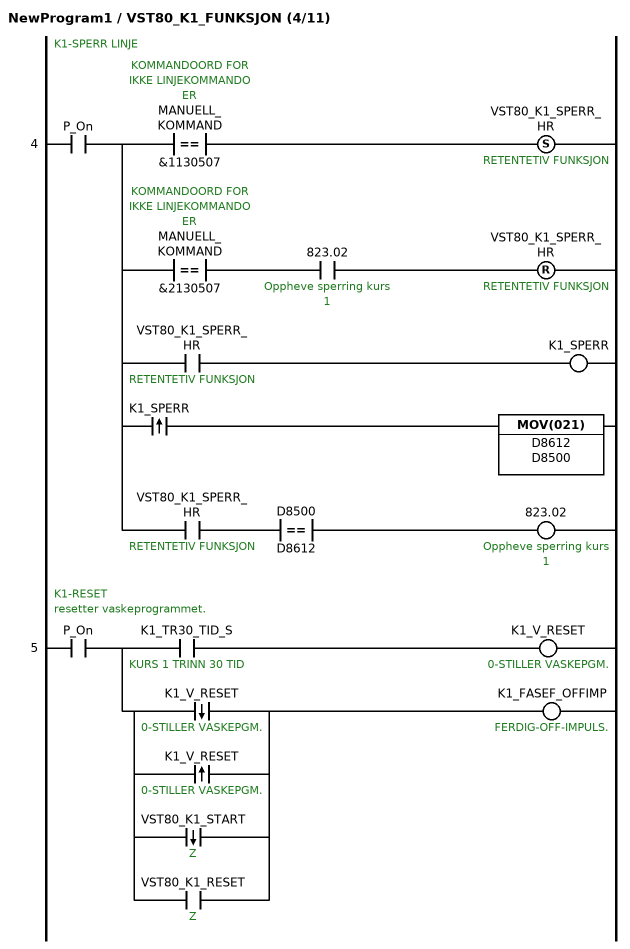
; [picture p120: NewProgram1 / VST80_K1_FUNKSJON, rungs 4-5]
; rung 4: K1-SPERR LINJE
LD P_On
OUT TR0
AND=L(301) MANUELL_KOMMAND &1130507  ; KOMMANDOORD FOR IKKE LINJEKOMMANDOER
SET VST80_K1_SPERR_HR  ; RETENTETIV FUNKSJON
LD TR0
AND=L(301) MANUELL_KOMMAND &2130507  ; KOMMANDOORD FOR IKKE LINJEKOMMANDOER
AND 823.02  ; Oppheve sperring kurs 1
RSET VST80_K1_SPERR_HR  ; RETENTETIV FUNKSJON
LD TR0
AND VST80_K1_SPERR_HR  ; RETENTETIV FUNKSJON
OUT K1_SPERR
LD TR0
@AND K1_SPERR
MOV(021) D8612 D8500
LD TR0
AND VST80_K1_SPERR_HR  ; RETENTETIV FUNKSJON
AND=(300) D8500 D8612
OUT 823.02  ; Oppheve sperring kurs 1
; rung 5: K1-RESET / resetter vaskeprogrammet.
LD P_On
OUT TR0
AND K1_TR30_TID_S  ; KURS 1 TRINN 30 TID
OUT K1_V_RESET  ; 0-STILLER VASKEPGM.
LD TR0
%LD K1_V_RESET  ; 0-STILLER VASKEPGM.
@OR K1_V_RESET  ; 0-STILLER VASKEPGM.
%OR VST80_K1_START  ; Z
OR VST80_K1_RESET  ; Z
ANDLD
OUT K1_FASEF_OFFIMP  ; FERDIG-OFF-IMPULS.

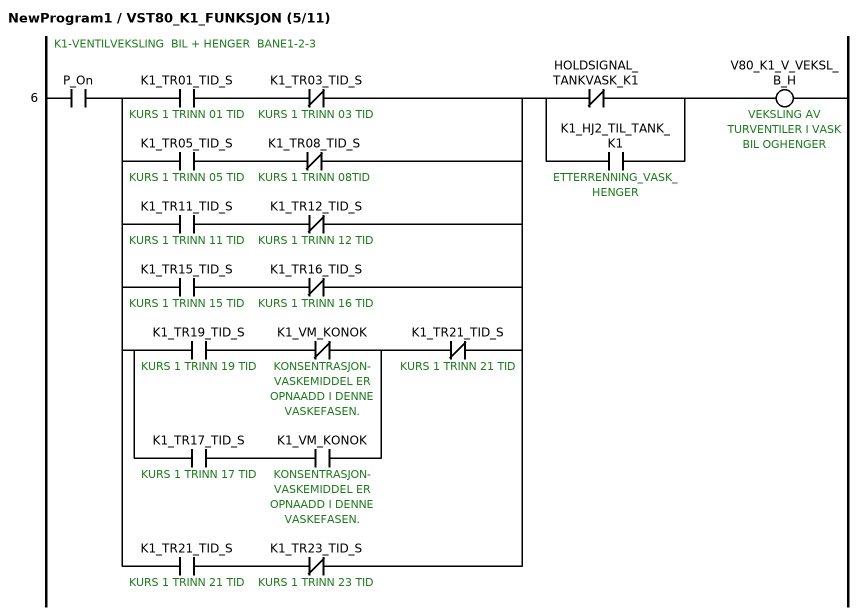
; rung 6: K1-VENTILVEKSLING  BIL + HENGER  BANE1-2-3
LD P_On
LD K1_TR01_TID_S  ; KURS 1 TRINN 01 TID
ANDNOT K1_TR03_TID_S  ; KURS 1 TRINN 03 TID
LD K1_TR05_TID_S  ; KURS 1 TRINN 05 TID
ANDNOT K1_TR08_TID_S  ; KURS 1 TRINN 08TID
ORLD
LD K1_TR11_TID_S  ; KURS 1 TRINN 11 TID
ANDNOT K1_TR12_TID_S  ; KURS 1 TRINN 12 TID
ORLD
LD K1_TR15_TID_S  ; KURS 1 TRINN 15 TID
ANDNOT K1_TR16_TID_S  ; KURS 1 TRINN 16 TID
ORLD
LD K1_TR19_TID_S  ; KURS 1 TRINN 19 TID
ANDNOT K1_VM_KONOK  ; KONSENTRASJON-VASKEMIDDEL ER OPNAADD I DENNE VASKEFASEN.
LD K1_TR17_TID_S  ; KURS 1 TRINN 17 TID
AND K1_VM_KONOK  ; KONSENTRASJON-VASKEMIDDEL ER OPNAADD I DENNE VASKEFASEN.
ORLD
ANDNOT K1_TR21_TID_S  ; KURS 1 TRINN 21 TID
ORLD
LD K1_TR21_TID_S  ; KURS 1 TRINN 21 TID
ANDNOT K1_TR23_TID_S  ; KURS 1 TRINN 23 TID
ORLD
ANDLD
LDNOT HOLDSIGNAL_TANKVASK_K1
OR K1_HJ2_TIL_TANK_K1  ; ETTERRENNING_VASK_HENGER
ANDLD
OUT V80_K1_V_VEKSL_B_H  ; VEKSLING AV TURVENTILER I VASK BIL OGHENGER

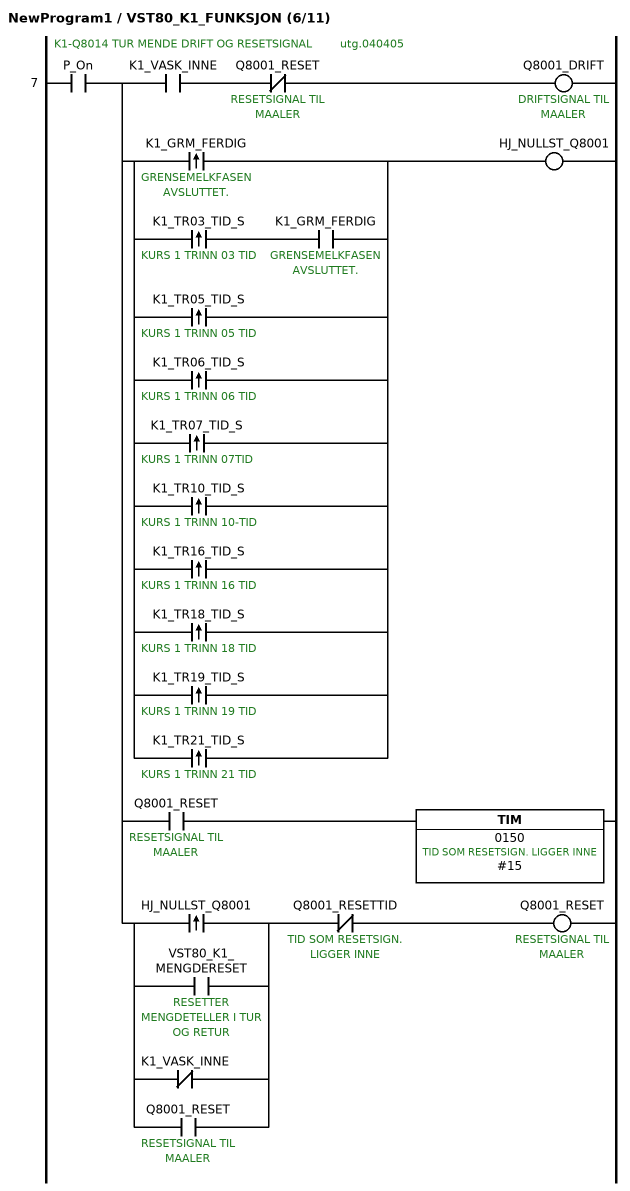
; rung 7: K1-Q8014 TUR MENDE DRIFT OG RESETSIGNAL        utg.040405
LD P_On
OUT TR0
AND K1_VASK_INNE
ANDNOT Q8001_RESET  ; RESETSIGNAL TIL MAALER
OUT Q8001_DRIFT  ; DRIFTSIGNAL TIL MAALER
LD TR0
@LD K1_GRM_FERDIG  ; GRENSEMELKFASEN AVSLUTTET.
@LD K1_TR03_TID_S  ; KURS 1 TRINN 03 TID
AND K1_GRM_FERDIG  ; GRENSEMELKFASEN AVSLUTTET.
ORLD
@OR K1_TR05_TID_S  ; KURS 1 TRINN 05 TID
@OR K1_TR06_TID_S  ; KURS 1 TRINN 06 TID
@OR K1_TR07_TID_S  ; KURS 1 TRINN 07TID
@OR K1_TR10_TID_S  ; KURS 1 TRINN 10-TID
@OR K1_TR16_TID_S  ; KURS 1 TRINN 16 TID
@OR K1_TR18_TID_S  ; KURS 1 TRINN 18 TID
@OR K1_TR19_TID_S  ; KURS 1 TRINN 19 TID
@OR K1_TR21_TID_S  ; KURS 1 TRINN 21 TID
ANDLD
OUT HJ_NULLST_Q8001
LD TR0
AND Q8001_RESET  ; RESETSIGNAL TIL MAALER
TIM 0150 #15  ; TID SOM RESETSIGN. LIGGER INNE
LD TR0
@LD HJ_NULLST_Q8001
OR VST80_K1_MENGDERESET  ; RESETTER MENGDETELLER I TUR OG RETUR
ORNOT K1_VASK_INNE
OR Q8001_RESET  ; RESETSIGNAL TIL MAALER
ANDLD
ANDNOT Q8001_RESETTID  ; TID SOM RESETSIGN. LIGGER INNE
OUT Q8001_RESET  ; RESETSIGNAL TIL MAALER

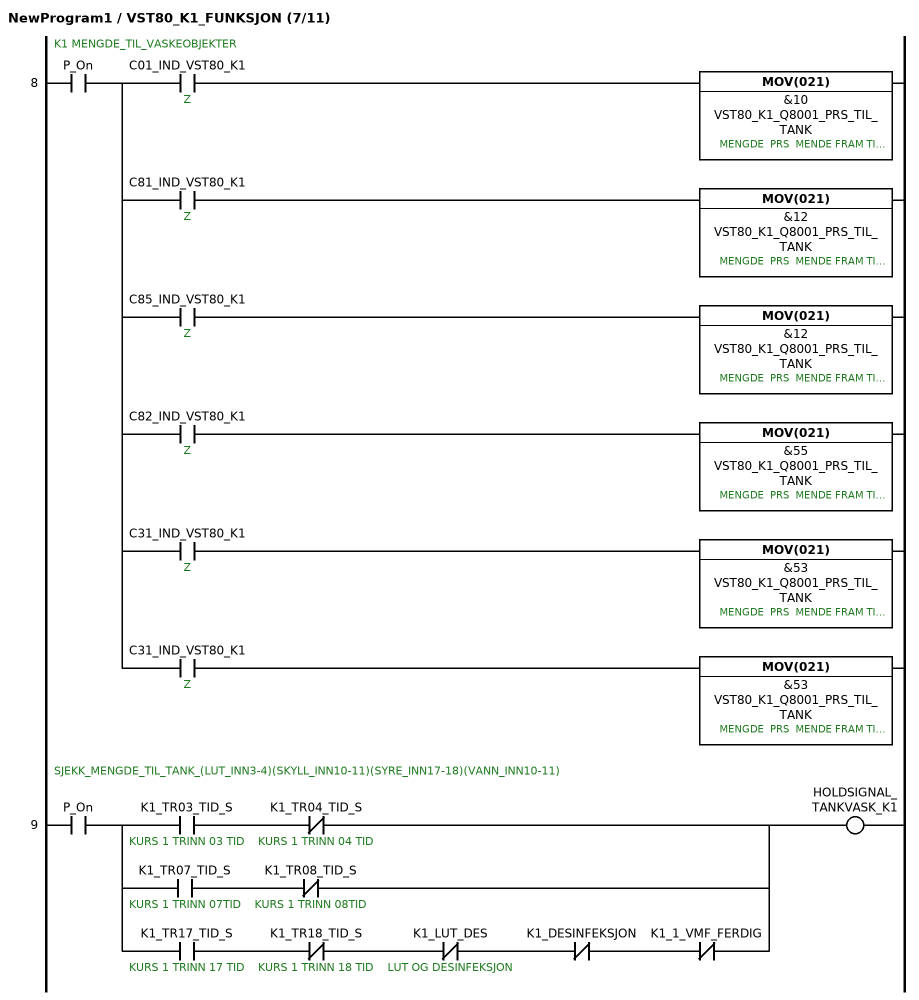
; rung 8: K1 MENGDE_TIL_VASKEOBJEKTER
LD P_On
OUT TR0
AND C01_IND_VST80_K1  ; Z
MOV(021) &10 VST80_K1_Q8001_PRS_TIL_TANK  ; MENGDE  PRS  MENDE FRAM TIL TANK
LD TR0
AND C81_IND_VST80_K1  ; Z
MOV(021) &12 VST80_K1_Q8001_PRS_TIL_TANK  ; MENGDE  PRS  MENDE FRAM TIL TANK
LD TR0
AND C85_IND_VST80_K1  ; Z
MOV(021) &12 VST80_K1_Q8001_PRS_TIL_TANK  ; MENGDE  PRS  MENDE FRAM TIL TANK
LD TR0
AND C82_IND_VST80_K1  ; Z
MOV(021) &55 VST80_K1_Q8001_PRS_TIL_TANK  ; MENGDE  PRS  MENDE FRAM TIL TANK
LD TR0
AND C31_IND_VST80_K1  ; Z
MOV(021) &53 VST80_K1_Q8001_PRS_TIL_TANK  ; MENGDE  PRS  MENDE FRAM TIL TANK
LD TR0
AND C31_IND_VST80_K1  ; Z
MOV(021) &53 VST80_K1_Q8001_PRS_TIL_TANK  ; MENGDE  PRS  MENDE FRAM TIL TANK
; rung 9: SJEKK_MENGDE_TIL_TANK_(LUT_INN3-4)(SKYLL_INN10-11)(SYRE_INN17-18)(VANN_INN10-11)
LD P_On
LD K1_TR03_TID_S  ; KURS 1 TRINN 03 TID
ANDNOT K1_TR04_TID_S  ; KURS 1 TRINN 04 TID
LD K1_TR07_TID_S  ; KURS 1 TRINN 07TID
ANDNOT K1_TR08_TID_S  ; KURS 1 TRINN 08TID
ORLD
LD K1_TR17_TID_S  ; KURS 1 TRINN 17 TID
ANDNOT K1_TR18_TID_S  ; KURS 1 TRINN 18 TID
ANDNOT K1_LUT_DES  ; LUT OG DESINFEKSJON
ANDNOT K1_DESINFEKSJON
ANDNOT K1_1_VMF_FERDIG
ORLD
ANDLD
OUT HOLDSIGNAL_TANKVASK_K1

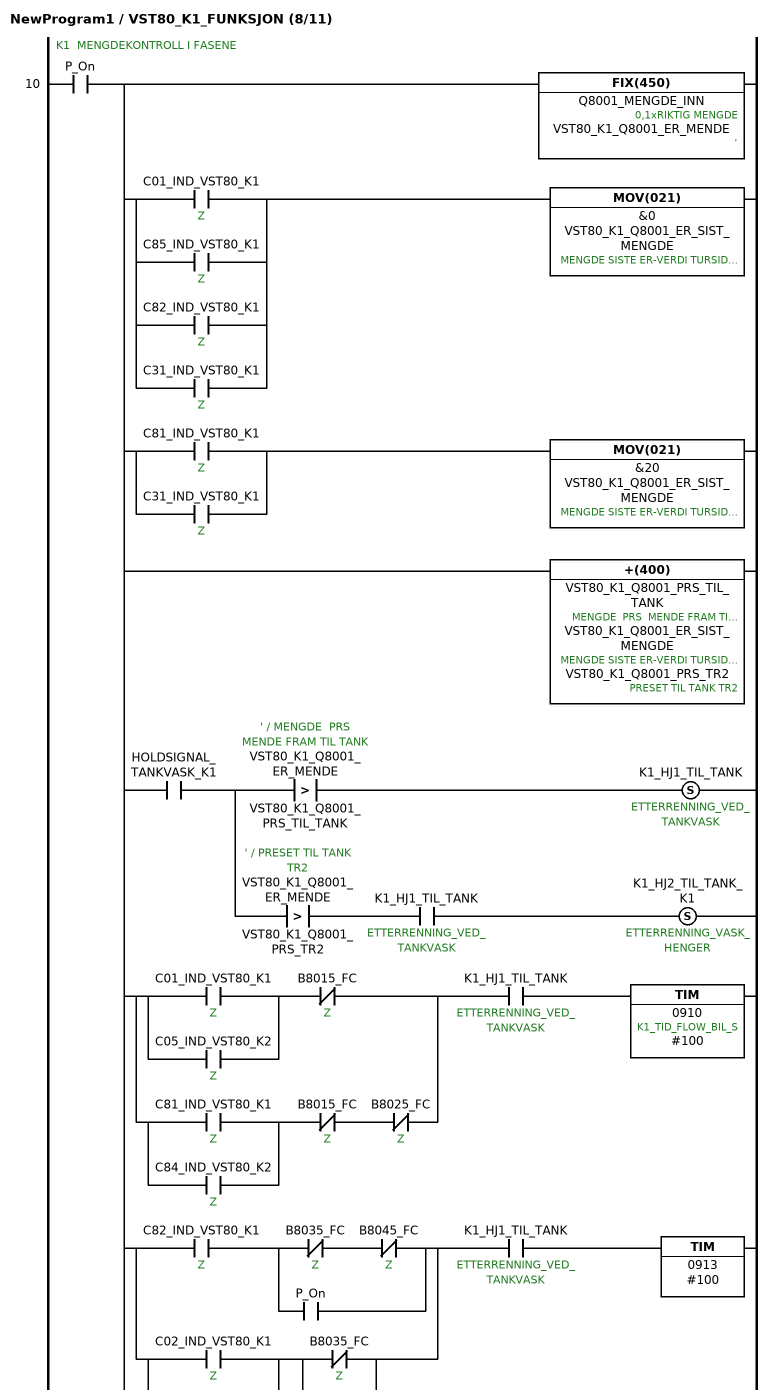

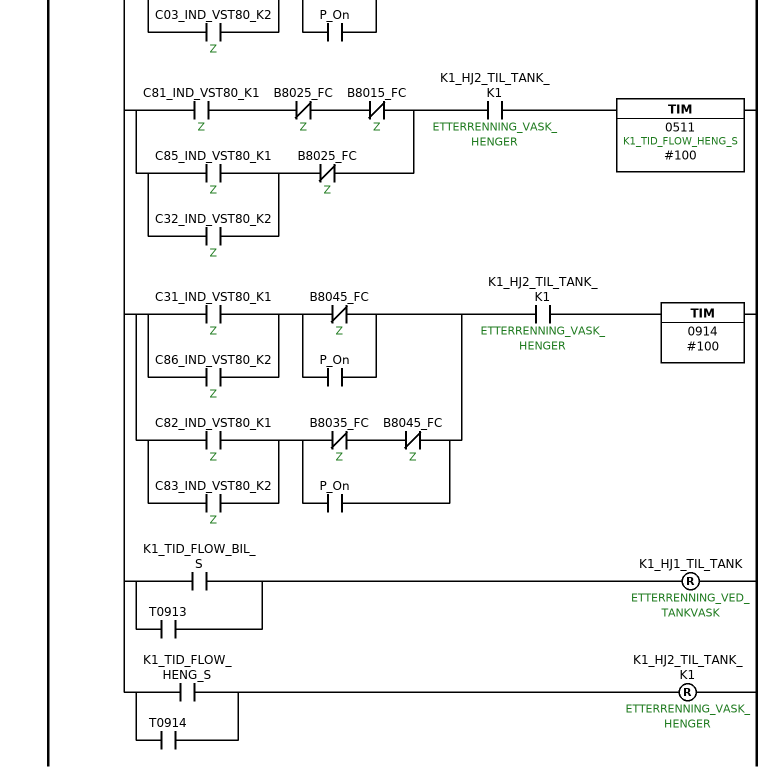
; rung 10: K1  MENGDEKONTROLL I FASENE
LD P_On
OUT TR0
FIX(450) Q8001_MENGDE_INN VST80_K1_Q8001_ER_MENDE  ; 0,1xRIKTIG MENGDE, '
LD C01_IND_VST80_K1  ; Z
OR C85_IND_VST80_K1  ; Z
OR C82_IND_VST80_K1  ; Z
OR C31_IND_VST80_K1  ; Z
ANDLD
MOV(021) &0 VST80_K1_Q8001_ER_SIST_MENGDE  ; MENGDE SISTE ER-VERDI TURSIDE PAA KURSEN
LD TR0
LD C81_IND_VST80_K1  ; Z
OR C31_IND_VST80_K1  ; Z
ANDLD
MOV(021) &20 VST80_K1_Q8001_ER_SIST_MENGDE  ; MENGDE SISTE ER-VERDI TURSIDE PAA KURSEN
LD TR0
+(400) VST80_K1_Q8001_PRS_TIL_TANK VST80_K1_Q8001_ER_SIST_MENGDE VST80_K1_Q8001_PRS_TR2  ; MENGDE  PRS  MENDE FRAM TIL TANK, MENGDE SISTE ER-VERDI TURSIDE PAA KURSEN, PRESET TIL TANK TR2
AND HOLDSIGNAL_TANKVASK_K1
OUT TR1
AND>(320) VST80_K1_Q8001_ER_MENDE VST80_K1_Q8001_PRS_TIL_TANK  ; ', MENGDE  PRS  MENDE FRAM TIL TANK
SET K1_HJ1_TIL_TANK  ; ETTERRENNING_VED_TANKVASK
LD TR1
AND>(320) VST80_K1_Q8001_ER_MENDE VST80_K1_Q8001_PRS_TR2  ; ', PRESET TIL TANK TR2
AND K1_HJ1_TIL_TANK  ; ETTERRENNING_VED_TANKVASK
SET K1_HJ2_TIL_TANK_K1  ; ETTERRENNING_VASK_HENGER
LD TR0
LD C01_IND_VST80_K1  ; Z
OR C05_IND_VST80_K2  ; Z
ANDNOT B8015_FC  ; Z
LD C81_IND_VST80_K1  ; Z
OR C84_IND_VST80_K2  ; Z
ANDNOT B8015_FC  ; Z
ANDNOT B8025_FC  ; Z
ORLD
ANDLD
AND K1_HJ1_TIL_TANK  ; ETTERRENNING_VED_TANKVASK
TIM 0910 #100  ; K1_TID_FLOW_BIL_S
LD TR0
LD C82_IND_VST80_K1  ; Z
LDNOT B8035_FC  ; Z
ANDNOT B8045_FC  ; Z
OR P_On
ANDLD
LD C02_IND_VST80_K1  ; Z
OR C03_IND_VST80_K2  ; Z
LDNOT B8035_FC  ; Z
OR P_On
ANDLD
ORLD
ANDLD
AND K1_HJ1_TIL_TANK  ; ETTERRENNING_VED_TANKVASK
TIM 0913 #100
LD TR0
LD C81_IND_VST80_K1  ; Z
ANDNOT B8025_FC  ; Z
ANDNOT B8015_FC  ; Z
LD C85_IND_VST80_K1  ; Z
OR C32_IND_VST80_K2  ; Z
ANDNOT B8025_FC  ; Z
ORLD
ANDLD
AND K1_HJ2_TIL_TANK_K1  ; ETTERRENNING_VASK_HENGER
TIM 0511 #100  ; K1_TID_FLOW_HENG_S
LD TR0
LD C31_IND_VST80_K1  ; Z
OR C86_IND_VST80_K2  ; Z
LDNOT B8045_FC  ; Z
OR P_On
ANDLD
LD C82_IND_VST80_K1  ; Z
OR C83_IND_VST80_K2  ; Z
LDNOT B8035_FC  ; Z
ANDNOT B8045_FC  ; Z
OR P_On
ANDLD
ORLD
ANDLD
AND K1_HJ2_TIL_TANK_K1  ; ETTERRENNING_VASK_HENGER
TIM 0914 #100
LD TR0
LD K1_TID_FLOW_BIL_S
OR T0913
ANDLD
RSET K1_HJ1_TIL_TANK  ; ETTERRENNING_VED_TANKVASK
LD TR0
LD K1_TID_FLOW_HENG_S
OR T0914
ANDLD
RSET K1_HJ2_TIL_TANK_K1  ; ETTERRENNING_VASK_HENGER

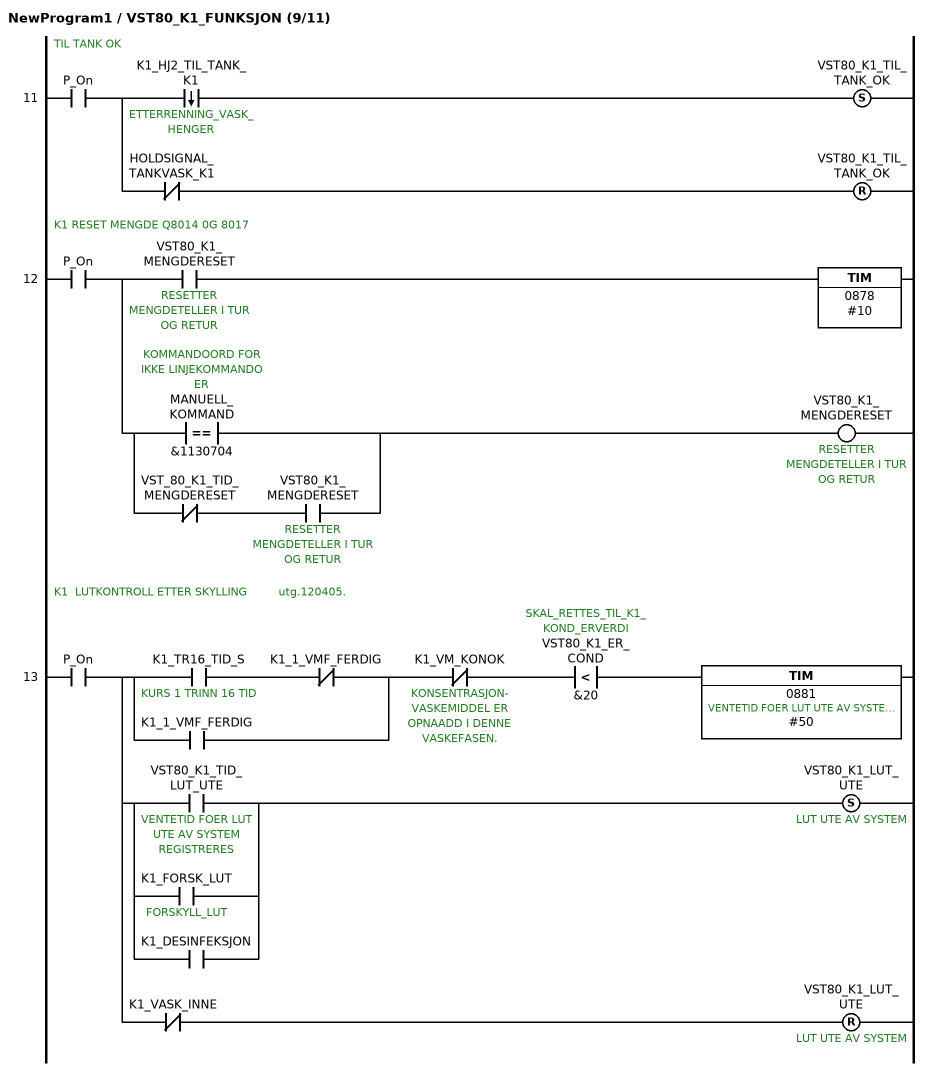
; rung 11: TIL TANK OK
LD P_On
OUT TR0
%AND K1_HJ2_TIL_TANK_K1  ; ETTERRENNING_VASK_HENGER
SET VST80_K1_TIL_TANK_OK
LD TR0
ANDNOT HOLDSIGNAL_TANKVASK_K1
RSET VST80_K1_TIL_TANK_OK
; rung 12: K1 RESET MENGDE Q8014 0G 8017
LD P_On
OUT TR0
AND VST80_K1_MENGDERESET  ; RESETTER MENGDETELLER I TUR OG RETUR
TIM 0878 #10
LD TR0
LD=L(301) MANUELL_KOMMAND &1130704  ; KOMMANDOORD FOR IKKE LINJEKOMMANDOER
LDNOT VST_80_K1_TID_MENGDERESET
AND VST80_K1_MENGDERESET  ; RESETTER MENGDETELLER I TUR OG RETUR
ORLD
ANDLD
OUT VST80_K1_MENGDERESET  ; RESETTER MENGDETELLER I TUR OG RETUR
; rung 13: K1  LUTKONTROLL ETTER SKYLLING         utg.120405.
LD P_On
OUT TR0
LD K1_TR16_TID_S  ; KURS 1 TRINN 16 TID
ANDNOT K1_1_VMF_FERDIG
OR K1_1_VMF_FERDIG
ANDLD
ANDNOT K1_VM_KONOK  ; KONSENTRASJON-VASKEMIDDEL ER OPNAADD I DENNE VASKEFASEN.
AND<(310) VST80_K1_ER_COND &20  ; SKAL_RETTES_TIL_K1_KOND_ERVERDI
TIM 0881 #50  ; VENTETID FOER LUT UTE AV SYSTEM REGISTRERES
LD TR0
LD VST80_K1_TID_LUT_UTE  ; VENTETID FOER LUT UTE AV SYSTEM REGISTRERES
OR K1_FORSK_LUT  ; FORSKYLL_LUT
OR K1_DESINFEKSJON
ANDLD
SET VST80_K1_LUT_UTE  ; LUT UTE AV SYSTEM
LD TR0
ANDNOT K1_VASK_INNE
RSET VST80_K1_LUT_UTE  ; LUT UTE AV SYSTEM

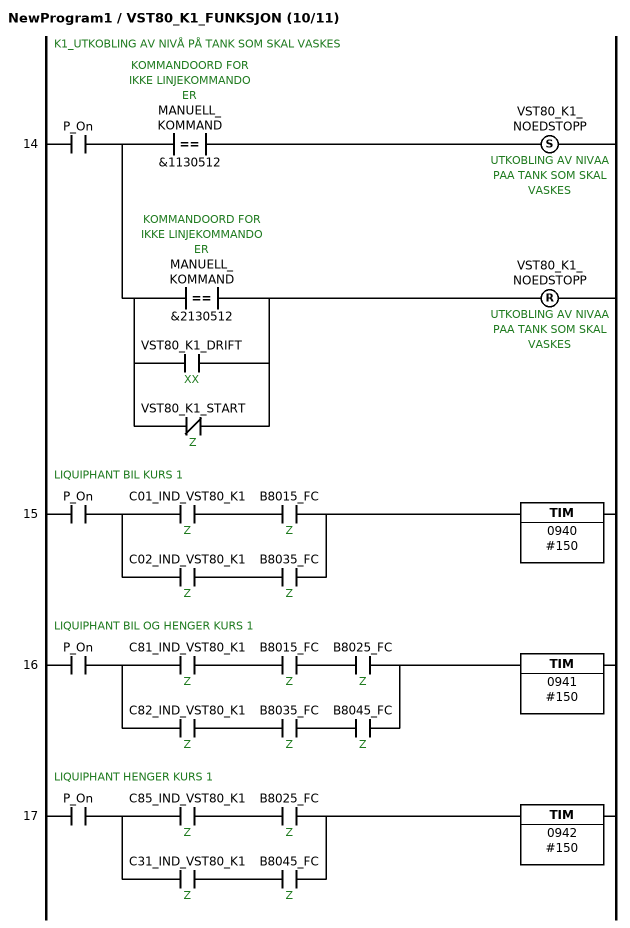
; rung 14: K1_UTKOBLING AV NIVÅ PÅ TANK SOM SKAL VASKES
LD P_On
OUT TR0
AND=L(301) MANUELL_KOMMAND &1130512  ; KOMMANDOORD FOR IKKE LINJEKOMMANDOER
SET VST80_K1_NOEDSTOPP  ; UTKOBLING AV NIVAA PAA TANK SOM SKAL VASKES
LD TR0
LD=L(301) MANUELL_KOMMAND &2130512  ; KOMMANDOORD FOR IKKE LINJEKOMMANDOER
OR VST80_K1_DRIFT  ; XX
ORNOT VST80_K1_START  ; Z
ANDLD
RSET VST80_K1_NOEDSTOPP  ; UTKOBLING AV NIVAA PAA TANK SOM SKAL VASKES
; rung 15: LIQUIPHANT BIL KURS 1
LD P_On
LD C01_IND_VST80_K1  ; Z
AND B8015_FC  ; Z
LD C02_IND_VST80_K1  ; Z
AND B8035_FC  ; Z
ORLD
ANDLD
TIM 0940 #150
; rung 16: LIQUIPHANT BIL OG HENGER KURS 1
LD P_On
LD C81_IND_VST80_K1  ; Z
AND B8015_FC  ; Z
AND B8025_FC  ; Z
LD C82_IND_VST80_K1  ; Z
AND B8035_FC  ; Z
AND B8045_FC  ; Z
ORLD
ANDLD
TIM 0941 #150
; rung 17: LIQUIPHANT HENGER KURS 1
LD P_On
LD C85_IND_VST80_K1  ; Z
AND B8025_FC  ; Z
LD C31_IND_VST80_K1  ; Z
AND B8045_FC  ; Z
ORLD
ANDLD
TIM 0942 #150

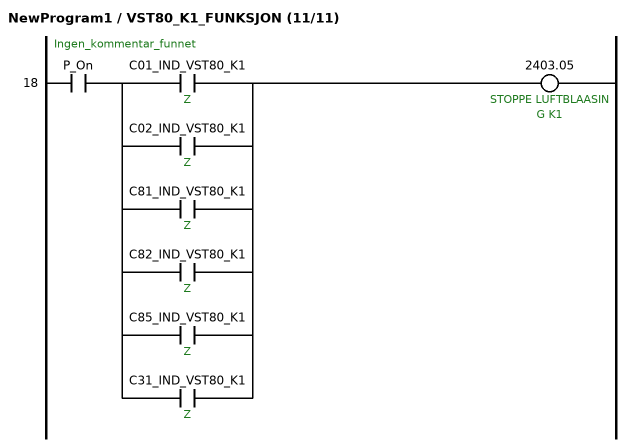
; rung 18: Ingen_kommentar_funnet
LD P_On
LD C01_IND_VST80_K1  ; Z
OR C02_IND_VST80_K1  ; Z
OR C81_IND_VST80_K1  ; Z
OR C82_IND_VST80_K1  ; Z
OR C85_IND_VST80_K1  ; Z
OR C31_IND_VST80_K1  ; Z
ANDLD
OUT 2403.05  ; STOPPE LUFTBLAASING K1
; rung 19: Ingen_kommentar_funnet

### Section VST80_K1_OBJEKTER
; Styring av objektene i kurs K1

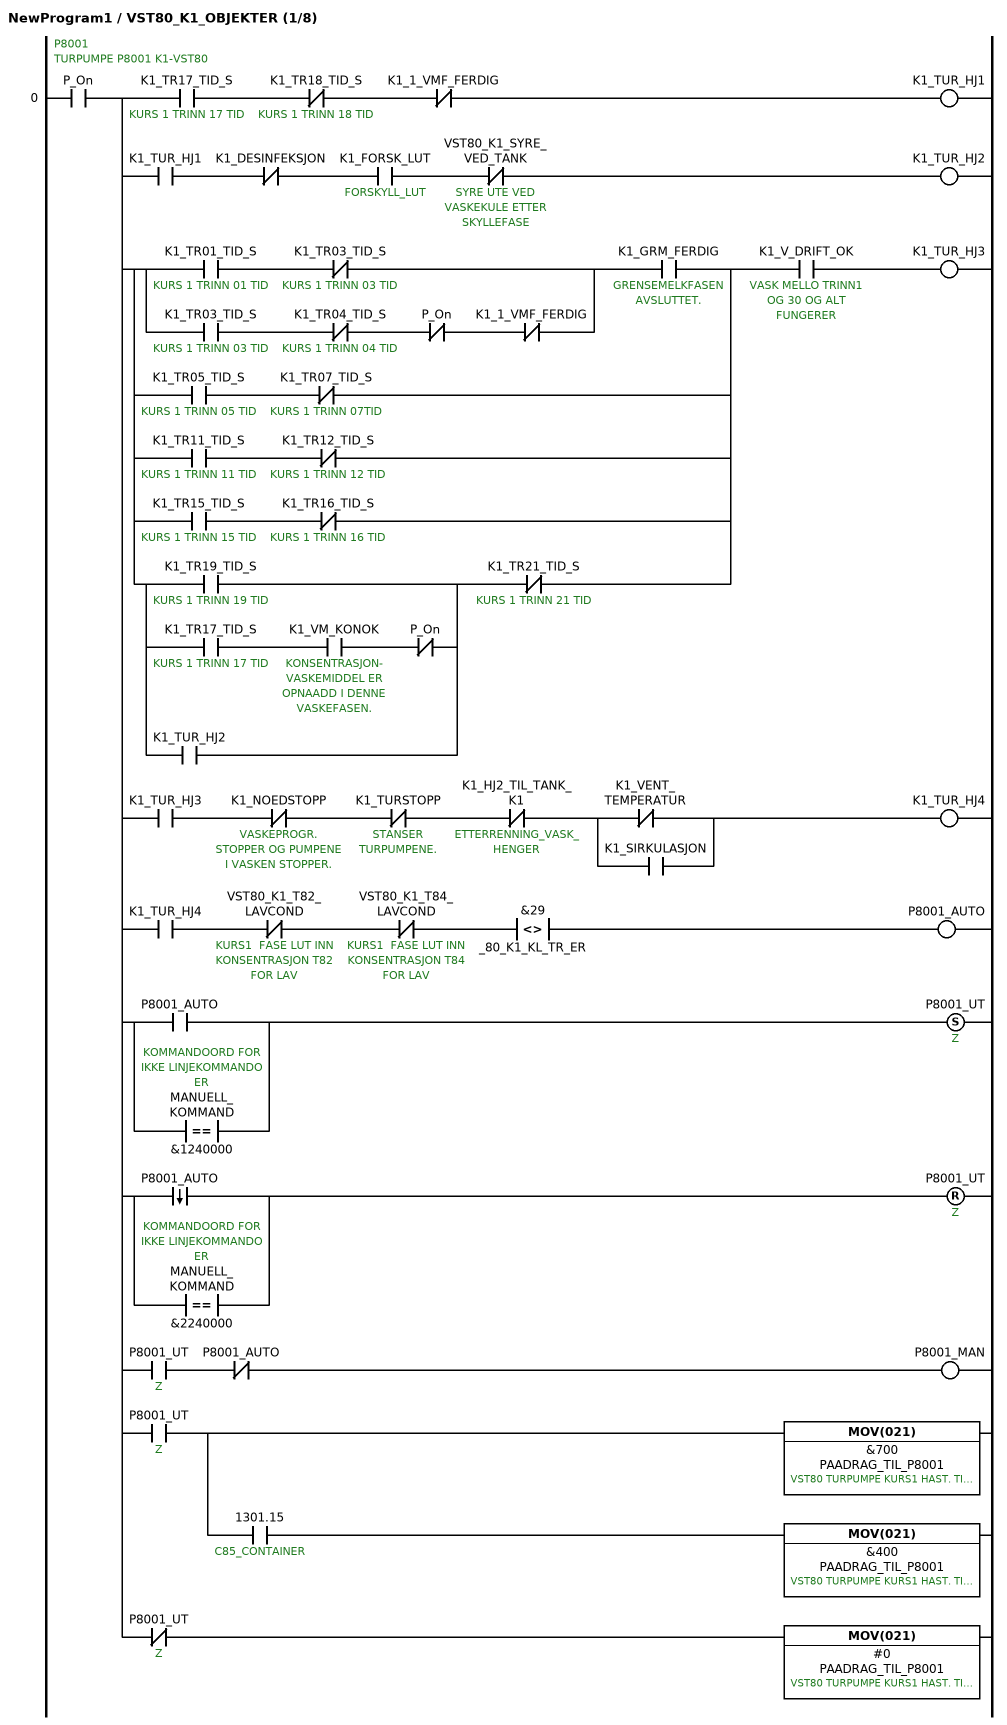
; rung 0: P8001 / TURPUMPE P8001 K1-VST80
LD P_On
OUT TR0
AND K1_TR17_TID_S  ; KURS 1 TRINN 17 TID
ANDNOT K1_TR18_TID_S  ; KURS 1 TRINN 18 TID
ANDNOT K1_1_VMF_FERDIG
OUT K1_TUR_HJ1
LD TR0
AND K1_TUR_HJ1
ANDNOT K1_DESINFEKSJON
AND K1_FORSK_LUT  ; FORSKYLL_LUT
ANDNOT VST80_K1_SYRE_VED_TANK  ; SYRE UTE VED VASKEKULE ETTER SKYLLEFASE
OUT K1_TUR_HJ2
LD TR0
LD K1_TR01_TID_S  ; KURS 1 TRINN 01 TID
ANDNOT K1_TR03_TID_S  ; KURS 1 TRINN 03 TID
LD K1_TR03_TID_S  ; KURS 1 TRINN 03 TID
ANDNOT K1_TR04_TID_S  ; KURS 1 TRINN 04 TID
ANDNOT P_On
ANDNOT K1_1_VMF_FERDIG
ORLD
AND K1_GRM_FERDIG  ; GRENSEMELKFASEN AVSLUTTET.
LD K1_TR05_TID_S  ; KURS 1 TRINN 05 TID
ANDNOT K1_TR07_TID_S  ; KURS 1 TRINN 07TID
ORLD
LD K1_TR11_TID_S  ; KURS 1 TRINN 11 TID
ANDNOT K1_TR12_TID_S  ; KURS 1 TRINN 12 TID
ORLD
LD K1_TR15_TID_S  ; KURS 1 TRINN 15 TID
ANDNOT K1_TR16_TID_S  ; KURS 1 TRINN 16 TID
ORLD
LD K1_TR19_TID_S  ; KURS 1 TRINN 19 TID
LD K1_TR17_TID_S  ; KURS 1 TRINN 17 TID
AND K1_VM_KONOK  ; KONSENTRASJON-VASKEMIDDEL ER OPNAADD I DENNE VASKEFASEN.
ANDNOT P_On
ORLD
OR K1_TUR_HJ2
ANDNOT K1_TR21_TID_S  ; KURS 1 TRINN 21 TID
ORLD
ANDLD
AND K1_V_DRIFT_OK  ; VASK MELLO TRINN1 OG 30 OG ALT FUNGERER
OUT K1_TUR_HJ3
LD TR0
AND K1_TUR_HJ3
ANDNOT K1_NOEDSTOPP  ; VASKEPROGR. STOPPER OG PUMPENE I VASKEN STOPPER.
ANDNOT K1_TURSTOPP  ; STANSER TURPUMPENE.
ANDNOT K1_HJ2_TIL_TANK_K1  ; ETTERRENNING_VASK_HENGER
LDNOT K1_VENT_TEMPERATUR
OR K1_SIRKULASJON
ANDLD
OUT K1_TUR_HJ4
LD TR0
AND K1_TUR_HJ4
ANDNOT VST80_K1_T82_LAVCOND  ; KURS1  FASE LUT INN KONSENTRASJON T82 FOR LAV
ANDNOT VST80_K1_T84_LAVCOND  ; KURS1  FASE LUT INN KONSENTRASJON T84 FOR LAV
AND<>(305) &29 _80_K1_KL_TR_ER
OUT P8001_AUTO
LD TR0
LD P8001_AUTO
OR=L(301) MANUELL_KOMMAND &1240000  ; KOMMANDOORD FOR IKKE LINJEKOMMANDOER
ANDLD
SET P8001_UT  ; Z
LD TR0
%LD P8001_AUTO
OR=L(301) MANUELL_KOMMAND &2240000  ; KOMMANDOORD FOR IKKE LINJEKOMMANDOER
ANDLD
RSET P8001_UT  ; Z
LD TR0
AND P8001_UT  ; Z
ANDNOT P8001_AUTO
OUT P8001_MAN
LD TR0
AND P8001_UT  ; Z
MOV(021) &700 PAADRAG_TIL_P8001  ; VST80 TURPUMPE KURS1 HAST. TIL FR.OMF. P8010
AND 1301.15  ; C85_CONTAINER
MOV(021) &400 PAADRAG_TIL_P8001  ; VST80 TURPUMPE KURS1 HAST. TIL FR.OMF. P8010
LD TR0
ANDNOT P8001_UT  ; Z
MOV(021) #0 PAADRAG_TIL_P8001  ; VST80 TURPUMPE KURS1 HAST. TIL FR.OMF. P8010

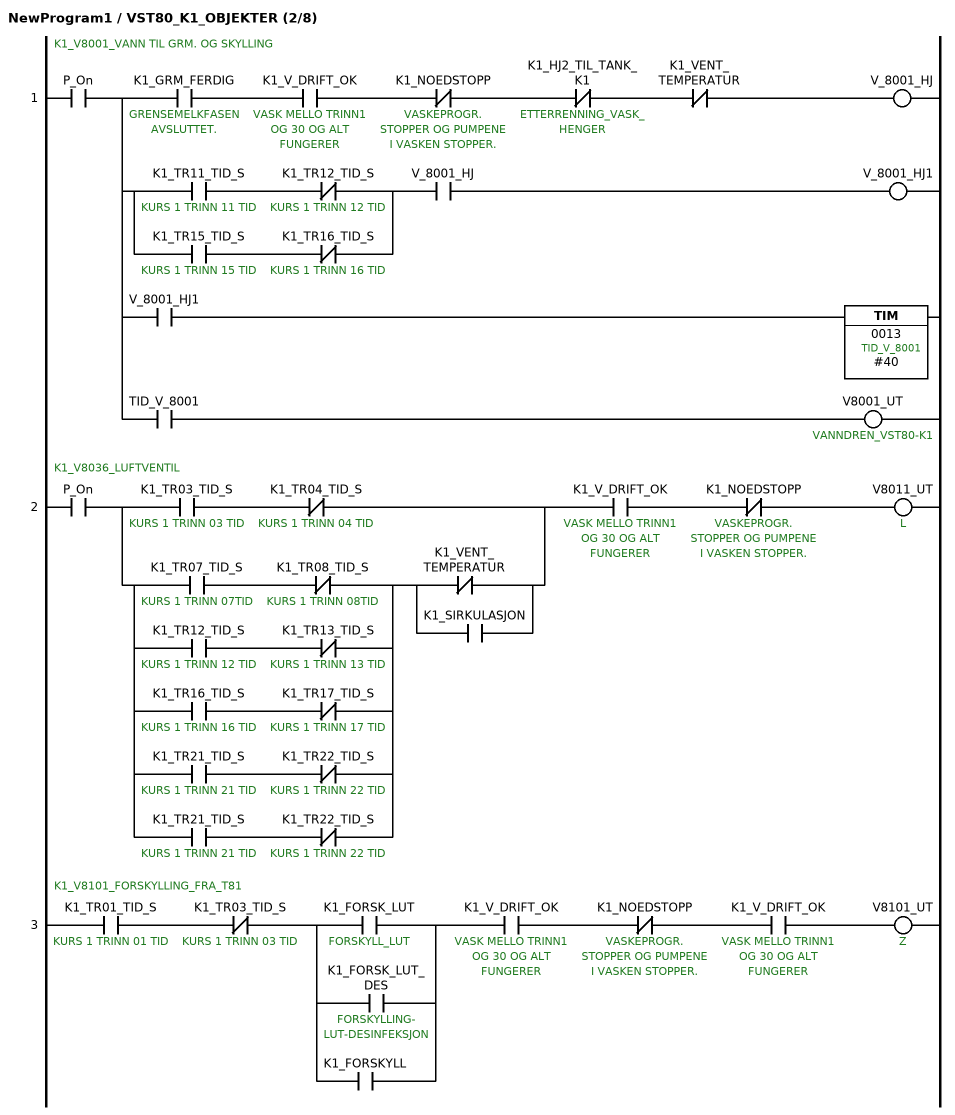
; rung 1: K1_V8001_VANN TIL GRM. OG SKYLLING
LD P_On
OUT TR0
AND K1_GRM_FERDIG  ; GRENSEMELKFASEN AVSLUTTET.
AND K1_V_DRIFT_OK  ; VASK MELLO TRINN1 OG 30 OG ALT FUNGERER
ANDNOT K1_NOEDSTOPP  ; VASKEPROGR. STOPPER OG PUMPENE I VASKEN STOPPER.
ANDNOT K1_HJ2_TIL_TANK_K1  ; ETTERRENNING_VASK_HENGER
ANDNOT K1_VENT_TEMPERATUR
OUT V_8001_HJ
LD TR0
LD K1_TR11_TID_S  ; KURS 1 TRINN 11 TID
ANDNOT K1_TR12_TID_S  ; KURS 1 TRINN 12 TID
LD K1_TR15_TID_S  ; KURS 1 TRINN 15 TID
ANDNOT K1_TR16_TID_S  ; KURS 1 TRINN 16 TID
ORLD
ANDLD
AND V_8001_HJ
OUT V_8001_HJ1
LD TR0
AND V_8001_HJ1
TIM 0013 #40  ; TID_V_8001
LD TR0
AND TID_V_8001
OUT V8001_UT  ; VANNDREN_VST80-K1
; rung 2: K1_V8036_LUFTVENTIL
LD P_On
LD K1_TR03_TID_S  ; KURS 1 TRINN 03 TID
ANDNOT K1_TR04_TID_S  ; KURS 1 TRINN 04 TID
LD K1_TR07_TID_S  ; KURS 1 TRINN 07TID
ANDNOT K1_TR08_TID_S  ; KURS 1 TRINN 08TID
LD K1_TR12_TID_S  ; KURS 1 TRINN 12 TID
ANDNOT K1_TR13_TID_S  ; KURS 1 TRINN 13 TID
ORLD
LD K1_TR16_TID_S  ; KURS 1 TRINN 16 TID
ANDNOT K1_TR17_TID_S  ; KURS 1 TRINN 17 TID
ORLD
LD K1_TR21_TID_S  ; KURS 1 TRINN 21 TID
ANDNOT K1_TR22_TID_S  ; KURS 1 TRINN 22 TID
ORLD
LD K1_TR21_TID_S  ; KURS 1 TRINN 21 TID
ANDNOT K1_TR22_TID_S  ; KURS 1 TRINN 22 TID
ORLD
LDNOT K1_VENT_TEMPERATUR
OR K1_SIRKULASJON
ANDLD
ORLD
ANDLD
AND K1_V_DRIFT_OK  ; VASK MELLO TRINN1 OG 30 OG ALT FUNGERER
ANDNOT K1_NOEDSTOPP  ; VASKEPROGR. STOPPER OG PUMPENE I VASKEN STOPPER.
OUT V8011_UT  ; L
; rung 3: K1_V8101_FORSKYLLING_FRA_T81
LD K1_TR01_TID_S  ; KURS 1 TRINN 01 TID
ANDNOT K1_TR03_TID_S  ; KURS 1 TRINN 03 TID
LD K1_FORSK_LUT  ; FORSKYLL_LUT
OR K1_FORSK_LUT_DES  ; FORSKYLLING- LUT-DESINFEKSJON
OR K1_FORSKYLL
ANDLD
AND K1_V_DRIFT_OK  ; VASK MELLO TRINN1 OG 30 OG ALT FUNGERER
ANDNOT K1_NOEDSTOPP  ; VASKEPROGR. STOPPER OG PUMPENE I VASKEN STOPPER.
AND K1_V_DRIFT_OK  ; VASK MELLO TRINN1 OG 30 OG ALT FUNGERER
OUT V8101_UT  ; Z

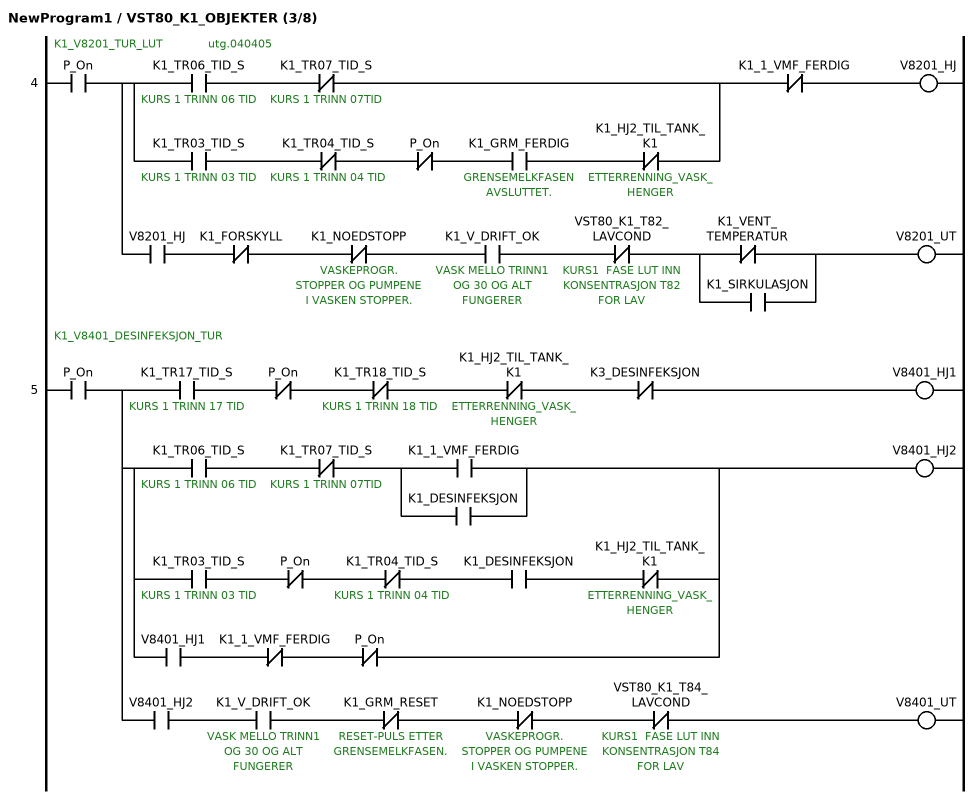
; rung 4: K1_V8201_TUR_LUT             utg.040405
LD P_On
OUT TR0
LD K1_TR06_TID_S  ; KURS 1 TRINN 06 TID
ANDNOT K1_TR07_TID_S  ; KURS 1 TRINN 07TID
LD K1_TR03_TID_S  ; KURS 1 TRINN 03 TID
ANDNOT K1_TR04_TID_S  ; KURS 1 TRINN 04 TID
ANDNOT P_On
AND K1_GRM_FERDIG  ; GRENSEMELKFASEN AVSLUTTET.
ANDNOT K1_HJ2_TIL_TANK_K1  ; ETTERRENNING_VASK_HENGER
ORLD
ANDLD
ANDNOT K1_1_VMF_FERDIG
OUT V8201_HJ
LD TR0
AND V8201_HJ
ANDNOT K1_FORSKYLL
ANDNOT K1_NOEDSTOPP  ; VASKEPROGR. STOPPER OG PUMPENE I VASKEN STOPPER.
AND K1_V_DRIFT_OK  ; VASK MELLO TRINN1 OG 30 OG ALT FUNGERER
ANDNOT VST80_K1_T82_LAVCOND  ; KURS1  FASE LUT INN KONSENTRASJON T82 FOR LAV
LDNOT K1_VENT_TEMPERATUR
OR K1_SIRKULASJON
ANDLD
OUT V8201_UT
; rung 5: K1_V8401_DESINFEKSJON_TUR
LD P_On
OUT TR0
AND K1_TR17_TID_S  ; KURS 1 TRINN 17 TID
ANDNOT P_On
ANDNOT K1_TR18_TID_S  ; KURS 1 TRINN 18 TID
ANDNOT K1_HJ2_TIL_TANK_K1  ; ETTERRENNING_VASK_HENGER
ANDNOT K3_DESINFEKSJON
OUT V8401_HJ1
LD TR0
LD K1_TR06_TID_S  ; KURS 1 TRINN 06 TID
ANDNOT K1_TR07_TID_S  ; KURS 1 TRINN 07TID
LD K1_1_VMF_FERDIG
OR K1_DESINFEKSJON
ANDLD
LD K1_TR03_TID_S  ; KURS 1 TRINN 03 TID
ANDNOT P_On
ANDNOT K1_TR04_TID_S  ; KURS 1 TRINN 04 TID
AND K1_DESINFEKSJON
ANDNOT K1_HJ2_TIL_TANK_K1  ; ETTERRENNING_VASK_HENGER
ORLD
LD V8401_HJ1
ANDNOT K1_1_VMF_FERDIG
ANDNOT P_On
ORLD
ANDLD
OUT V8401_HJ2
LD TR0
AND V8401_HJ2
AND K1_V_DRIFT_OK  ; VASK MELLO TRINN1 OG 30 OG ALT FUNGERER
ANDNOT K1_GRM_RESET  ; RESET-PULS ETTER GRENSEMELKFASEN.
ANDNOT K1_NOEDSTOPP  ; VASKEPROGR. STOPPER OG PUMPENE I VASKEN STOPPER.
ANDNOT VST80_K1_T84_LAVCOND  ; KURS1  FASE LUT INN KONSENTRASJON T84 FOR LAV
OUT V8401_UT

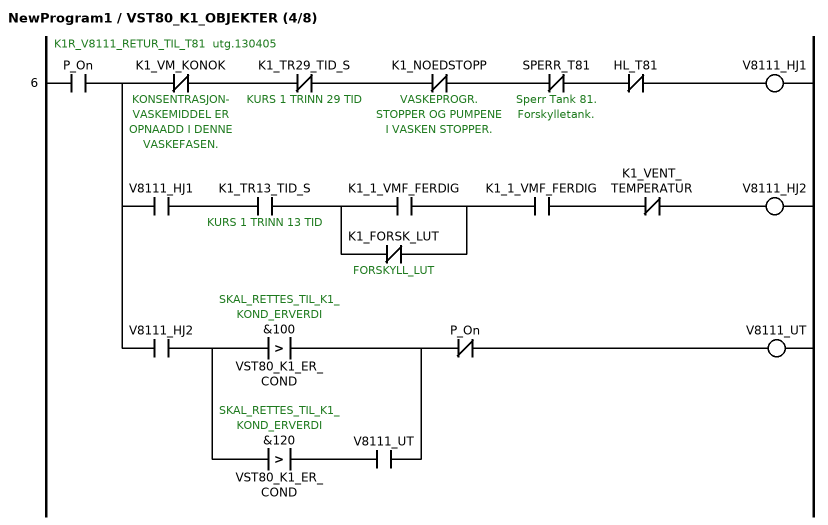
; rung 6: K1R_V8111_RETUR_TIL_T81  utg.130405
LD P_On
OUT TR0
ANDNOT K1_VM_KONOK  ; KONSENTRASJON-VASKEMIDDEL ER OPNAADD I DENNE VASKEFASEN.
ANDNOT K1_TR29_TID_S  ; KURS 1 TRINN 29 TID
ANDNOT K1_NOEDSTOPP  ; VASKEPROGR. STOPPER OG PUMPENE I VASKEN STOPPER.
ANDNOT SPERR_T81  ; Sperr Tank 81. Forskylletank.
ANDNOT HL_T81
OUT V8111_HJ1
LD TR0
AND V8111_HJ1
AND K1_TR13_TID_S  ; KURS 1 TRINN 13 TID
LD K1_1_VMF_FERDIG
ORNOT K1_FORSK_LUT  ; FORSKYLL_LUT
ANDLD
AND K1_1_VMF_FERDIG
ANDNOT K1_VENT_TEMPERATUR
OUT V8111_HJ2
LD TR0
AND V8111_HJ2
LD>(320) &100 VST80_K1_ER_COND  ; SKAL_RETTES_TIL_K1_KOND_ERVERDI
LD>(320) &120 VST80_K1_ER_COND  ; SKAL_RETTES_TIL_K1_KOND_ERVERDI
AND V8111_UT
ORLD
ANDLD
ANDNOT P_On
OUT V8111_UT

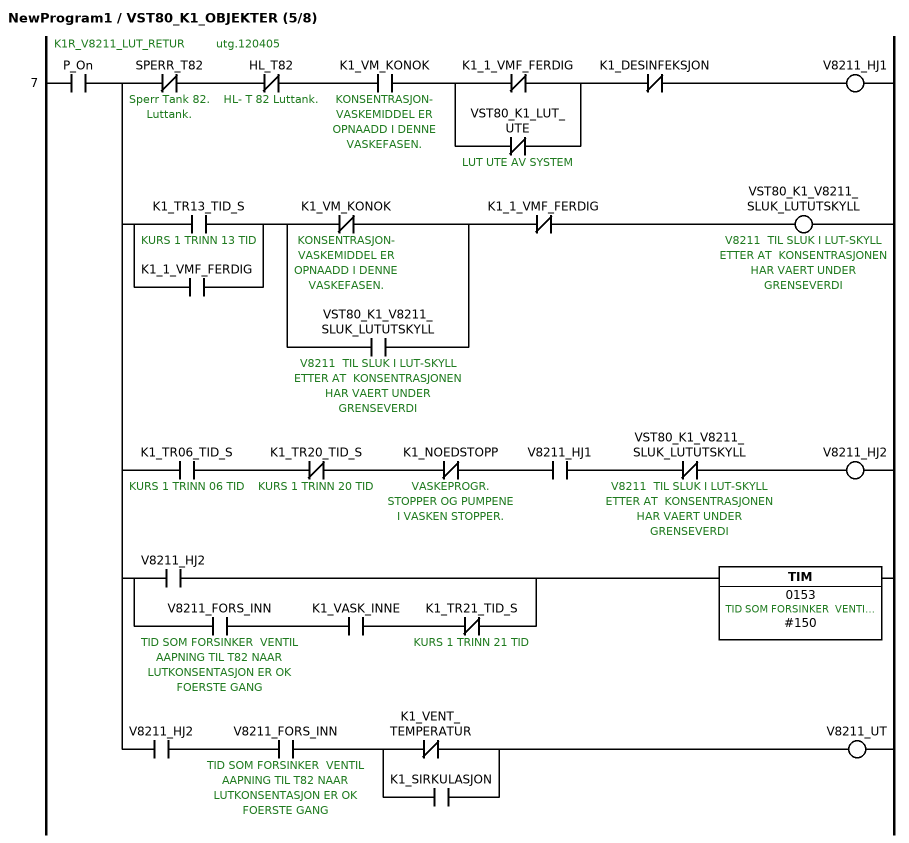
; rung 7: K1R_V8211_LUT_RETUR         utg.120405
LD P_On
OUT TR0
ANDNOT SPERR_T82  ; Sperr Tank 82. Luttank.
ANDNOT HL_T82  ; HL- T 82 Luttank.
AND K1_VM_KONOK  ; KONSENTRASJON-VASKEMIDDEL ER OPNAADD I DENNE VASKEFASEN.
LDNOT K1_1_VMF_FERDIG
ORNOT VST80_K1_LUT_UTE  ; LUT UTE AV SYSTEM
ANDLD
ANDNOT K1_DESINFEKSJON
OUT V8211_HJ1
LD TR0
LD K1_TR13_TID_S  ; KURS 1 TRINN 13 TID
OR K1_1_VMF_FERDIG
ANDLD
LDNOT K1_VM_KONOK  ; KONSENTRASJON-VASKEMIDDEL ER OPNAADD I DENNE VASKEFASEN.
OR VST80_K1_V8211_SLUK_LUTUTSKYLL  ; V8211  TIL SLUK I LUT-SKYLL ETTER AT  KONSENTRASJONEN HAR VAERT UNDER  GRENSEVERDI
ANDLD
ANDNOT K1_1_VMF_FERDIG
OUT VST80_K1_V8211_SLUK_LUTUTSKYLL  ; V8211  TIL SLUK I LUT-SKYLL ETTER AT  KONSENTRASJONEN HAR VAERT UNDER  GRENSEVERDI
LD TR0
AND K1_TR06_TID_S  ; KURS 1 TRINN 06 TID
ANDNOT K1_TR20_TID_S  ; KURS 1 TRINN 20 TID
ANDNOT K1_NOEDSTOPP  ; VASKEPROGR. STOPPER OG PUMPENE I VASKEN STOPPER.
AND V8211_HJ1
ANDNOT VST80_K1_V8211_SLUK_LUTUTSKYLL  ; V8211  TIL SLUK I LUT-SKYLL ETTER AT  KONSENTRASJONEN HAR VAERT UNDER  GRENSEVERDI
OUT V8211_HJ2
LD TR0
LD V8211_HJ2
LD V8211_FORS_INN  ; TID SOM FORSINKER  VENTIL AAPNING TIL T82 NAAR LUTKONSENTASJON ER OK FOERSTE GANG
AND K1_VASK_INNE
ANDNOT K1_TR21_TID_S  ; KURS 1 TRINN 21 TID
ORLD
ANDLD
TIM 0153 #150  ; TID SOM FORSINKER  VENTIL AAPNING TIL T82 NAAR LUTKONSENTASJON ER OK FOERSTE GANG
LD TR0
AND V8211_HJ2
AND V8211_FORS_INN  ; TID SOM FORSINKER  VENTIL AAPNING TIL T82 NAAR LUTKONSENTASJON ER OK FOERSTE GANG
LDNOT K1_VENT_TEMPERATUR
OR K1_SIRKULASJON
ANDLD
OUT V8211_UT

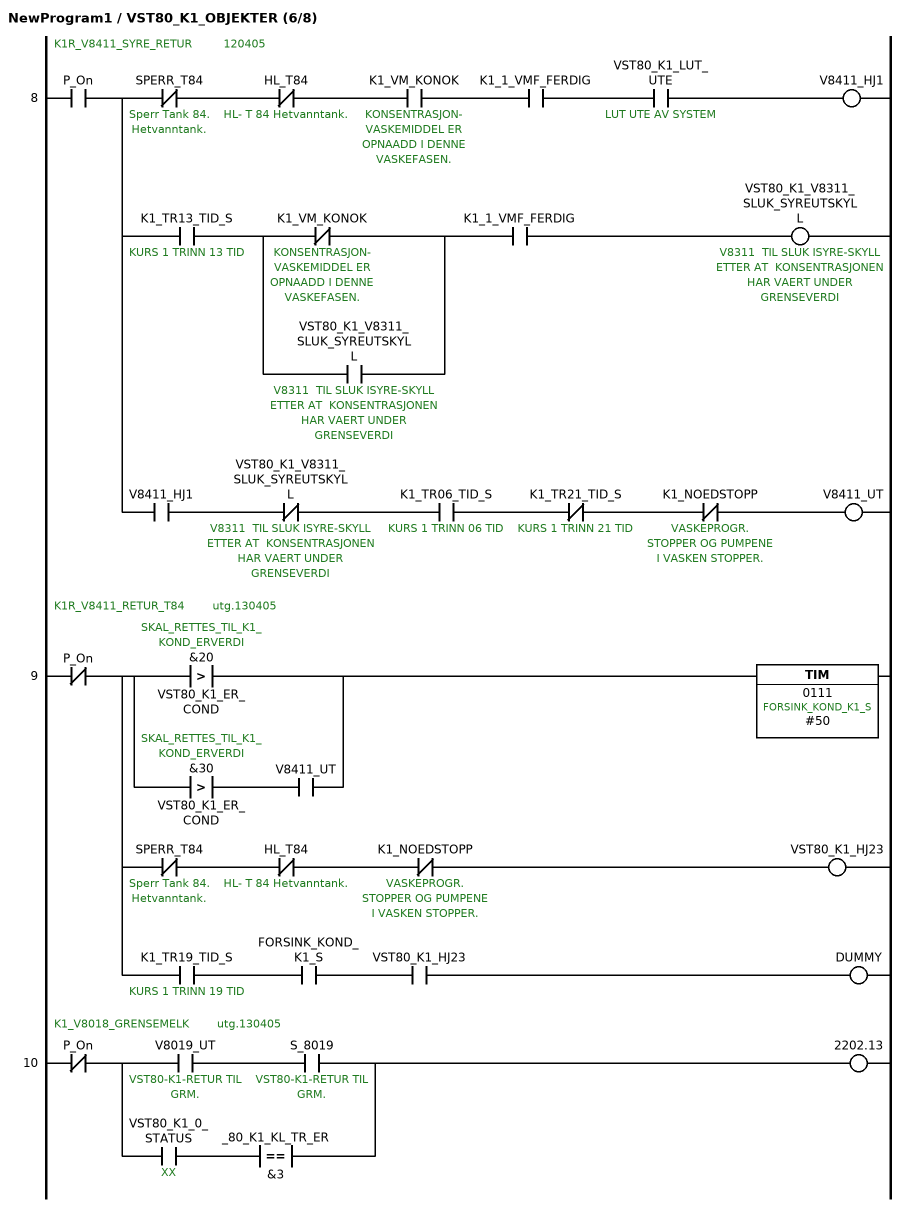
; rung 8: K1R_V8411_SYRE_RETUR         120405
LD P_On
OUT TR0
ANDNOT SPERR_T84  ; Sperr Tank 84. Hetvanntank.
ANDNOT HL_T84  ; HL- T 84 Hetvanntank.
AND K1_VM_KONOK  ; KONSENTRASJON-VASKEMIDDEL ER OPNAADD I DENNE VASKEFASEN.
AND K1_1_VMF_FERDIG
AND VST80_K1_LUT_UTE  ; LUT UTE AV SYSTEM
OUT V8411_HJ1
LD TR0
AND K1_TR13_TID_S  ; KURS 1 TRINN 13 TID
LDNOT K1_VM_KONOK  ; KONSENTRASJON-VASKEMIDDEL ER OPNAADD I DENNE VASKEFASEN.
OR VST80_K1_V8311_SLUK_SYREUTSKYLL  ; V8311  TIL SLUK ISYRE-SKYLL ETTER AT  KONSENTRASJONEN HAR VAERT UNDER  GRENSEVERDI
ANDLD
AND K1_1_VMF_FERDIG
OUT VST80_K1_V8311_SLUK_SYREUTSKYLL  ; V8311  TIL SLUK ISYRE-SKYLL ETTER AT  KONSENTRASJONEN HAR VAERT UNDER  GRENSEVERDI
LD TR0
AND V8411_HJ1
ANDNOT VST80_K1_V8311_SLUK_SYREUTSKYLL  ; V8311  TIL SLUK ISYRE-SKYLL ETTER AT  KONSENTRASJONEN HAR VAERT UNDER  GRENSEVERDI
AND K1_TR06_TID_S  ; KURS 1 TRINN 06 TID
ANDNOT K1_TR21_TID_S  ; KURS 1 TRINN 21 TID
ANDNOT K1_NOEDSTOPP  ; VASKEPROGR. STOPPER OG PUMPENE I VASKEN STOPPER.
OUT V8411_UT
; rung 9: K1R_V8411_RETUR_T84        utg.130405
LDNOT P_On
OUT TR0
LD>(320) &20 VST80_K1_ER_COND  ; SKAL_RETTES_TIL_K1_KOND_ERVERDI
LD>(320) &30 VST80_K1_ER_COND  ; SKAL_RETTES_TIL_K1_KOND_ERVERDI
AND V8411_UT
ORLD
ANDLD
TIM 0111 #50  ; FORSINK_KOND_K1_S
LD TR0
ANDNOT SPERR_T84  ; Sperr Tank 84. Hetvanntank.
ANDNOT HL_T84  ; HL- T 84 Hetvanntank.
ANDNOT K1_NOEDSTOPP  ; VASKEPROGR. STOPPER OG PUMPENE I VASKEN STOPPER.
OUT VST80_K1_HJ23
LD TR0
AND K1_TR19_TID_S  ; KURS 1 TRINN 19 TID
AND FORSINK_KOND_K1_S
AND VST80_K1_HJ23
OUT DUMMY
; rung 10: K1_V8018_GRENSEMELK        utg.130405
LDNOT P_On
LD V8019_UT  ; VST80-K1-RETUR TIL GRM.
AND S_8019  ; VST80-K1-RETUR TIL GRM.
LD VST80_K1_0_STATUS  ; XX
AND=(300) _80_K1_KL_TR_ER &3
ORLD
ANDLD
OUT 2202.13

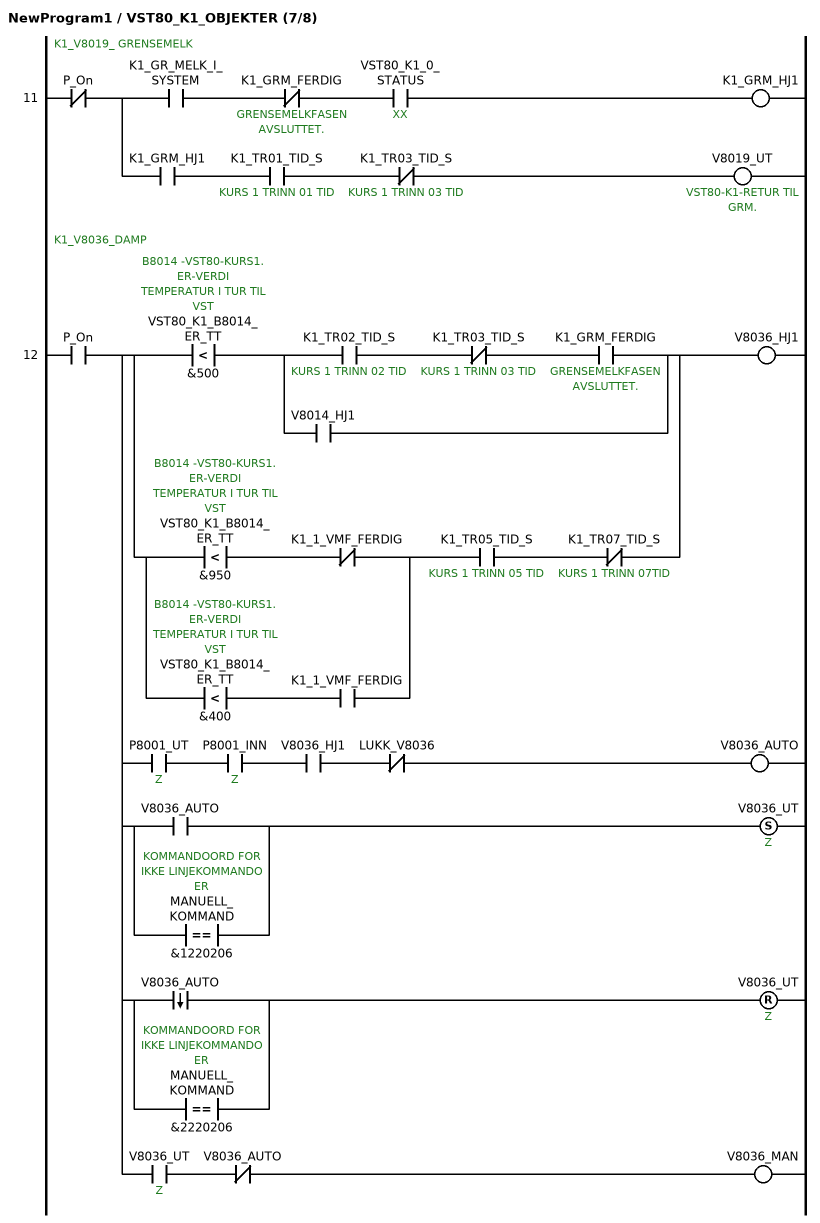
; rung 11: K1_V8019_GRENSEMELK
LDNOT P_On
OUT TR0
AND K1_GR_MELK_I_SYSTEM
ANDNOT K1_GRM_FERDIG  ; GRENSEMELKFASEN AVSLUTTET.
AND VST80_K1_0_STATUS  ; XX
OUT K1_GRM_HJ1
LD TR0
AND K1_GRM_HJ1
AND K1_TR01_TID_S  ; KURS 1 TRINN 01 TID
ANDNOT K1_TR03_TID_S  ; KURS 1 TRINN 03 TID
OUT V8019_UT  ; VST80-K1-RETUR TIL GRM.
; rung 12: K1_V8036_DAMP
LD P_On
OUT TR0
LD<(310) VST80_K1_B8014_ER_TT &500  ; B8014 -VST80-KURS1. ER-VERDI TEMPERATUR I TUR TIL VST
LD K1_TR02_TID_S  ; KURS 1 TRINN 02 TID
ANDNOT K1_TR03_TID_S  ; KURS 1 TRINN 03 TID
AND K1_GRM_FERDIG  ; GRENSEMELKFASEN AVSLUTTET.
OR V8014_HJ1
ANDLD
LD<(310) VST80_K1_B8014_ER_TT &950  ; B8014 -VST80-KURS1. ER-VERDI TEMPERATUR I TUR TIL VST
ANDNOT K1_1_VMF_FERDIG
LD<(310) VST80_K1_B8014_ER_TT &400  ; B8014 -VST80-KURS1. ER-VERDI TEMPERATUR I TUR TIL VST
AND K1_1_VMF_FERDIG
ORLD
AND K1_TR05_TID_S  ; KURS 1 TRINN 05 TID
ANDNOT K1_TR07_TID_S  ; KURS 1 TRINN 07TID
ORLD
ANDLD
OUT V8036_HJ1
LD TR0
AND P8001_UT  ; Z
AND P8001_INN  ; Z
AND V8036_HJ1
ANDNOT LUKK_V8036
OUT V8036_AUTO
LD TR0
LD V8036_AUTO
OR=L(301) MANUELL_KOMMAND &1220206  ; KOMMANDOORD FOR IKKE LINJEKOMMANDOER
ANDLD
SET V8036_UT  ; Z
LD TR0
%LD V8036_AUTO
OR=L(301) MANUELL_KOMMAND &2220206  ; KOMMANDOORD FOR IKKE LINJEKOMMANDOER
ANDLD
RSET V8036_UT  ; Z
LD TR0
AND V8036_UT  ; Z
ANDNOT V8036_AUTO
OUT V8036_MAN

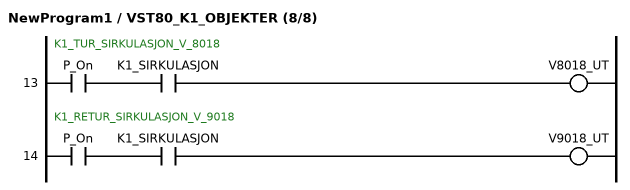
; rung 13: K1_TUR_SIRKULASJON_V_8018
LD P_On
AND K1_SIRKULASJON
OUT V8018_UT
; rung 14: K1_RETUR_SIRKULASJON_V_9018
LD P_On
AND K1_SIRKULASJON
OUT V9018_UT
; rung 15: Ingen_kommentar_funnet

### Section VST80_K1_KLAPRING
; VST80-KURS1 KLAPREPROGRAM

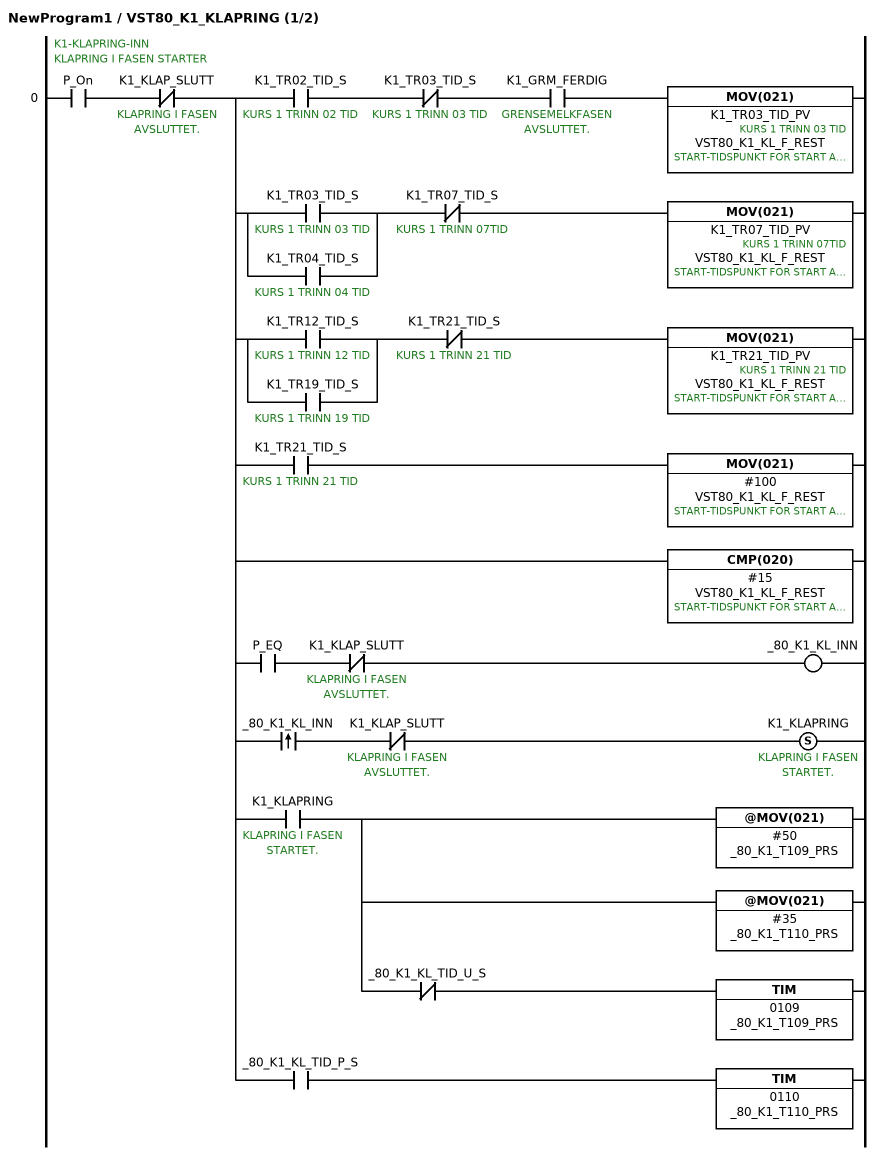
; rung 0: K1-KLAPRING-INN / KLAPRING I FASEN STARTER
LD P_On
ANDNOT K1_KLAP_SLUTT  ; KLAPRING I FASEN AVSLUTTET.
OUT TR0
AND K1_TR02_TID_S  ; KURS 1 TRINN 02 TID
ANDNOT K1_TR03_TID_S  ; KURS 1 TRINN 03 TID
AND K1_GRM_FERDIG  ; GRENSEMELKFASEN AVSLUTTET.
MOV(021) K1_TR03_TID_PV VST80_K1_KL_F_REST  ; KURS 1 TRINN 03 TID, START-TIDSPUNKT FOR START AV KLAPRING
LD TR0
LD K1_TR03_TID_S  ; KURS 1 TRINN 03 TID
OR K1_TR04_TID_S  ; KURS 1 TRINN 04 TID
ANDLD
ANDNOT K1_TR07_TID_S  ; KURS 1 TRINN 07TID
MOV(021) K1_TR07_TID_PV VST80_K1_KL_F_REST  ; KURS 1 TRINN 07TID, START-TIDSPUNKT FOR START AV KLAPRING
LD TR0
LD K1_TR12_TID_S  ; KURS 1 TRINN 12 TID
OR K1_TR19_TID_S  ; KURS 1 TRINN 19 TID
ANDLD
ANDNOT K1_TR21_TID_S  ; KURS 1 TRINN 21 TID
MOV(021) K1_TR21_TID_PV VST80_K1_KL_F_REST  ; KURS 1 TRINN 21 TID, START-TIDSPUNKT FOR START AV KLAPRING
LD TR0
AND K1_TR21_TID_S  ; KURS 1 TRINN 21 TID
MOV(021) #100 VST80_K1_KL_F_REST  ; START-TIDSPUNKT FOR START AV KLAPRING
LD TR0
CMP(020) #15 VST80_K1_KL_F_REST  ; START-TIDSPUNKT FOR START AV KLAPRING
AND P_EQ
ANDNOT K1_KLAP_SLUTT  ; KLAPRING I FASEN AVSLUTTET.
OUT _80_K1_KL_INN
LD TR0
@AND _80_K1_KL_INN
ANDNOT K1_KLAP_SLUTT  ; KLAPRING I FASEN AVSLUTTET.
SET K1_KLAPRING  ; KLAPRING I FASEN STARTET.
LD TR0
AND K1_KLAPRING  ; KLAPRING I FASEN STARTET.
@MOV(021) #50 _80_K1_T109_PRS
@MOV(021) #35 _80_K1_T110_PRS
ANDNOT _80_K1_KL_TID_U_S
TIM 0109 _80_K1_T109_PRS
LD TR0
AND _80_K1_KL_TID_P_S
TIM 0110 _80_K1_T110_PRS

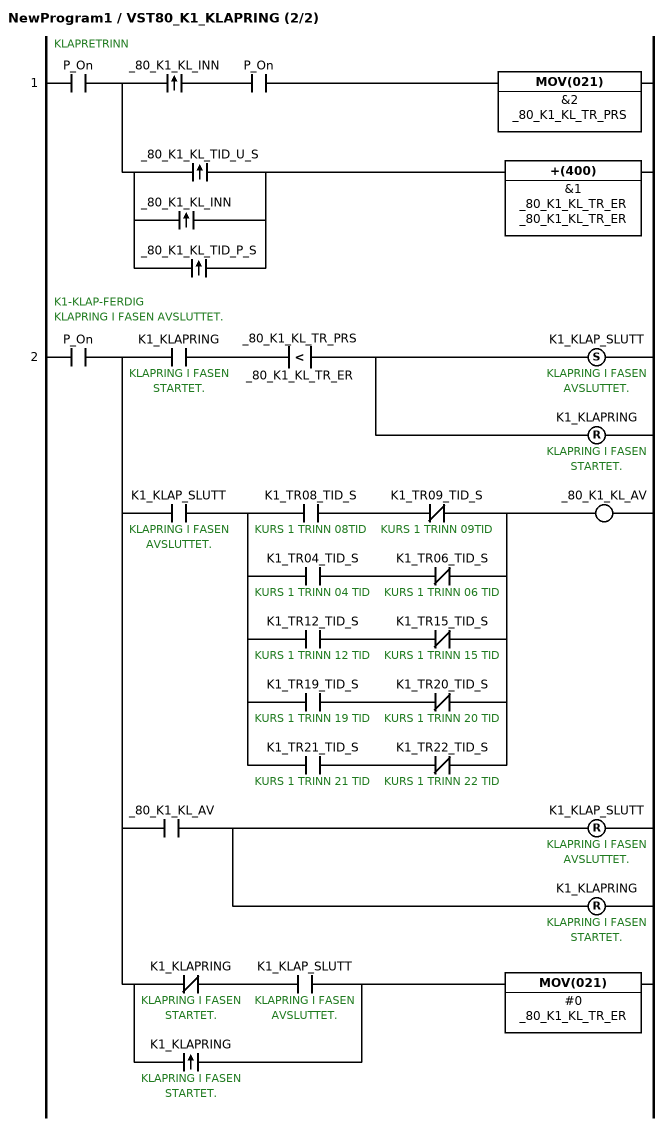
; rung 1: KLAPRETRINN
LD P_On
OUT TR0
@AND _80_K1_KL_INN
AND P_On
MOV(021) &2 _80_K1_KL_TR_PRS
LD TR0
@LD _80_K1_KL_TID_U_S
@OR _80_K1_KL_INN
@OR _80_K1_KL_TID_P_S
ANDLD
+(400) &1 _80_K1_KL_TR_ER _80_K1_KL_TR_ER
; rung 2: K1-KLAP-FERDIG / KLAPRING I FASEN AVSLUTTET.
LD P_On
OUT TR0
AND K1_KLAPRING  ; KLAPRING I FASEN STARTET.
AND<(310) _80_K1_KL_TR_PRS _80_K1_KL_TR_ER
SET K1_KLAP_SLUTT  ; KLAPRING I FASEN AVSLUTTET.
RSET K1_KLAPRING  ; KLAPRING I FASEN STARTET.
LD TR0
AND K1_KLAP_SLUTT  ; KLAPRING I FASEN AVSLUTTET.
LD K1_TR08_TID_S  ; KURS 1 TRINN 08TID
ANDNOT K1_TR09_TID_S  ; KURS 1 TRINN 09TID
LD K1_TR04_TID_S  ; KURS 1 TRINN 04 TID
ANDNOT K1_TR06_TID_S  ; KURS 1 TRINN 06 TID
ORLD
LD K1_TR12_TID_S  ; KURS 1 TRINN 12 TID
ANDNOT K1_TR15_TID_S  ; KURS 1 TRINN 15 TID
ORLD
LD K1_TR19_TID_S  ; KURS 1 TRINN 19 TID
ANDNOT K1_TR20_TID_S  ; KURS 1 TRINN 20 TID
ORLD
LD K1_TR21_TID_S  ; KURS 1 TRINN 21 TID
ANDNOT K1_TR22_TID_S  ; KURS 1 TRINN 22 TID
ORLD
ANDLD
OUT _80_K1_KL_AV
LD TR0
AND _80_K1_KL_AV
RSET K1_KLAP_SLUTT  ; KLAPRING I FASEN AVSLUTTET.
RSET K1_KLAPRING  ; KLAPRING I FASEN STARTET.
LD TR0
LDNOT K1_KLAPRING  ; KLAPRING I FASEN STARTET.
AND K1_KLAP_SLUTT  ; KLAPRING I FASEN AVSLUTTET.
@OR K1_KLAPRING  ; KLAPRING I FASEN STARTET.
ANDLD
MOV(021) #0 _80_K1_KL_TR_ER
; rung 3: Ingen_kommentar_funnet

### Section VST80_K1_GRAF_TR_
; OVERFØRING AV TRINN I VASK TIL GRAFIKK

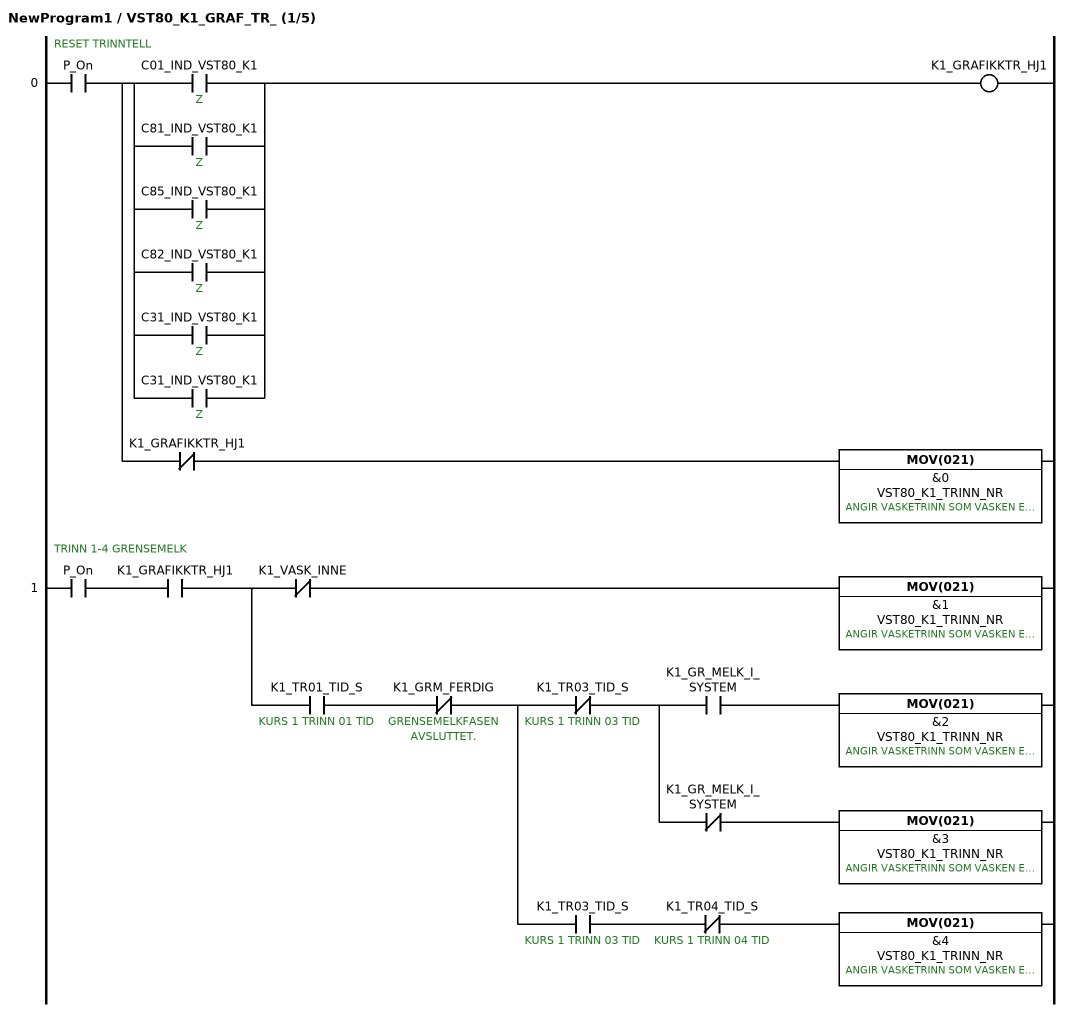
; rung 0: RESET TRINNTELL
LD P_On
OUT TR0
LD C01_IND_VST80_K1  ; Z
OR C81_IND_VST80_K1  ; Z
OR C85_IND_VST80_K1  ; Z
OR C82_IND_VST80_K1  ; Z
OR C31_IND_VST80_K1  ; Z
OR C31_IND_VST80_K1  ; Z
ANDLD
OUT K1_GRAFIKKTR_HJ1
LD TR0
ANDNOT K1_GRAFIKKTR_HJ1
MOV(021) &0 VST80_K1_TRINN_NR  ; ANGIR VASKETRINN SOM VASKEN ER I
; rung 1: TRINN 1-4 GRENSEMELK
LD P_On
AND K1_GRAFIKKTR_HJ1
OUT TR0
ANDNOT K1_VASK_INNE
MOV(021) &1 VST80_K1_TRINN_NR  ; ANGIR VASKETRINN SOM VASKEN ER I
LD TR0
AND K1_TR01_TID_S  ; KURS 1 TRINN 01 TID
ANDNOT K1_GRM_FERDIG  ; GRENSEMELKFASEN AVSLUTTET.
OUT TR0
ANDNOT K1_TR03_TID_S  ; KURS 1 TRINN 03 TID
OUT TR1
AND K1_GR_MELK_I_SYSTEM
MOV(021) &2 VST80_K1_TRINN_NR  ; ANGIR VASKETRINN SOM VASKEN ER I
LD TR1
ANDNOT K1_GR_MELK_I_SYSTEM
MOV(021) &3 VST80_K1_TRINN_NR  ; ANGIR VASKETRINN SOM VASKEN ER I
LD TR0
AND K1_TR03_TID_S  ; KURS 1 TRINN 03 TID
ANDNOT K1_TR04_TID_S  ; KURS 1 TRINN 04 TID
MOV(021) &4 VST80_K1_TRINN_NR  ; ANGIR VASKETRINN SOM VASKEN ER I

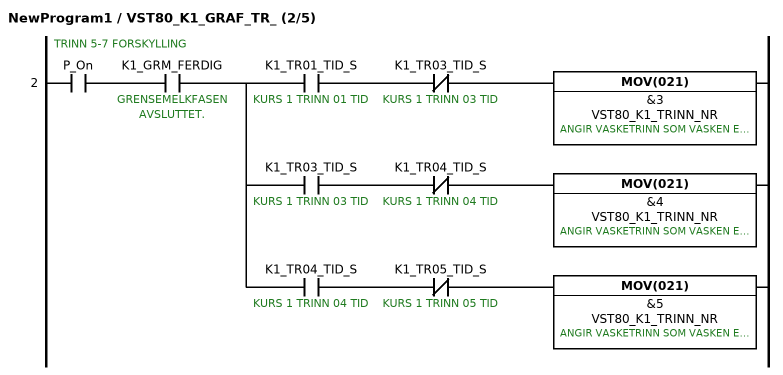
; rung 2: TRINN 5-7 FORSKYLLING
LD P_On
AND K1_GRM_FERDIG  ; GRENSEMELKFASEN AVSLUTTET.
OUT TR0
AND K1_TR01_TID_S  ; KURS 1 TRINN 01 TID
ANDNOT K1_TR03_TID_S  ; KURS 1 TRINN 03 TID
MOV(021) &3 VST80_K1_TRINN_NR  ; ANGIR VASKETRINN SOM VASKEN ER I
LD TR0
AND K1_TR03_TID_S  ; KURS 1 TRINN 03 TID
ANDNOT K1_TR04_TID_S  ; KURS 1 TRINN 04 TID
MOV(021) &4 VST80_K1_TRINN_NR  ; ANGIR VASKETRINN SOM VASKEN ER I
LD TR0
AND K1_TR04_TID_S  ; KURS 1 TRINN 04 TID
ANDNOT K1_TR05_TID_S  ; KURS 1 TRINN 05 TID
MOV(021) &5 VST80_K1_TRINN_NR  ; ANGIR VASKETRINN SOM VASKEN ER I

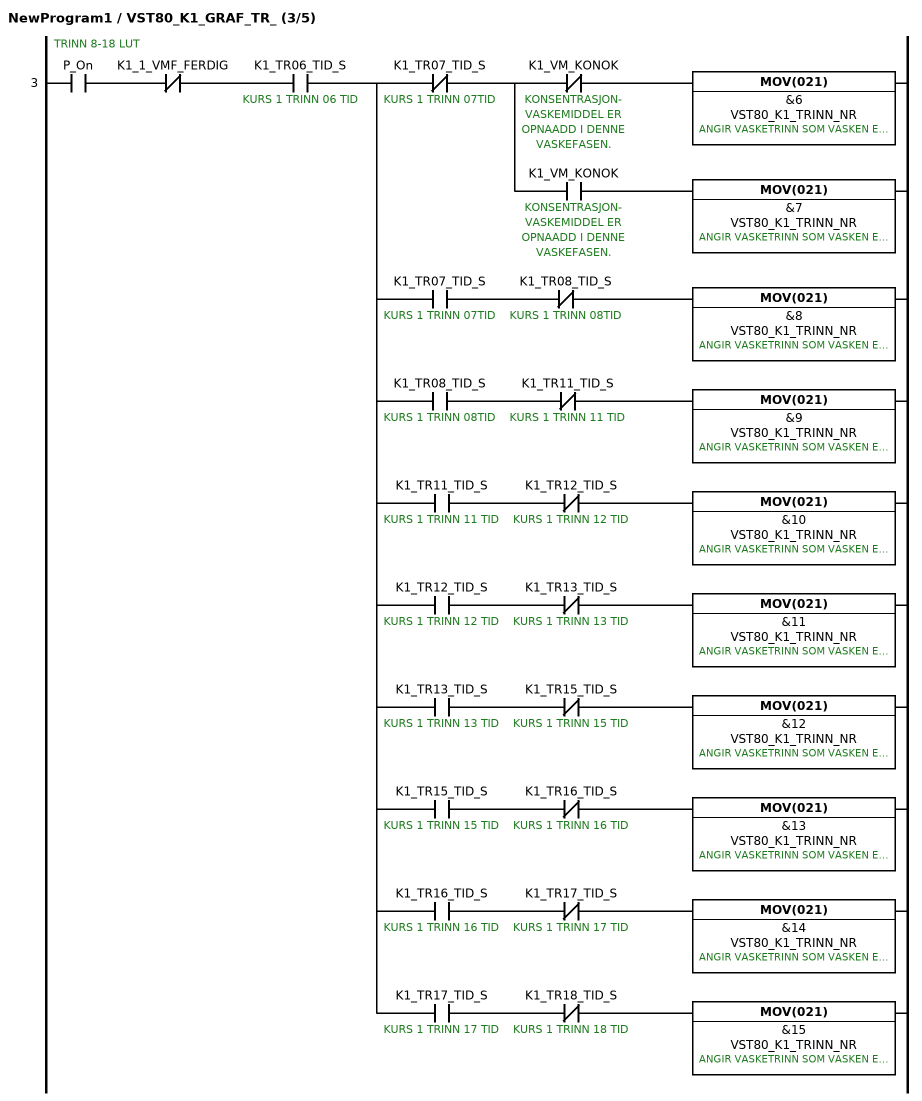
; rung 3: TRINN 8-18 LUT
LD P_On
ANDNOT K1_1_VMF_FERDIG
AND K1_TR06_TID_S  ; KURS 1 TRINN 06 TID
OUT TR0
ANDNOT K1_TR07_TID_S  ; KURS 1 TRINN 07TID
OUT TR1
ANDNOT K1_VM_KONOK  ; KONSENTRASJON-VASKEMIDDEL ER OPNAADD I DENNE VASKEFASEN.
MOV(021) &6 VST80_K1_TRINN_NR  ; ANGIR VASKETRINN SOM VASKEN ER I
LD TR1
AND K1_VM_KONOK  ; KONSENTRASJON-VASKEMIDDEL ER OPNAADD I DENNE VASKEFASEN.
MOV(021) &7 VST80_K1_TRINN_NR  ; ANGIR VASKETRINN SOM VASKEN ER I
LD TR0
AND K1_TR07_TID_S  ; KURS 1 TRINN 07TID
ANDNOT K1_TR08_TID_S  ; KURS 1 TRINN 08TID
MOV(021) &8 VST80_K1_TRINN_NR  ; ANGIR VASKETRINN SOM VASKEN ER I
LD TR0
AND K1_TR08_TID_S  ; KURS 1 TRINN 08TID
ANDNOT K1_TR11_TID_S  ; KURS 1 TRINN 11 TID
MOV(021) &9 VST80_K1_TRINN_NR  ; ANGIR VASKETRINN SOM VASKEN ER I
LD TR0
AND K1_TR11_TID_S  ; KURS 1 TRINN 11 TID
ANDNOT K1_TR12_TID_S  ; KURS 1 TRINN 12 TID
MOV(021) &10 VST80_K1_TRINN_NR  ; ANGIR VASKETRINN SOM VASKEN ER I
LD TR0
AND K1_TR12_TID_S  ; KURS 1 TRINN 12 TID
ANDNOT K1_TR13_TID_S  ; KURS 1 TRINN 13 TID
MOV(021) &11 VST80_K1_TRINN_NR  ; ANGIR VASKETRINN SOM VASKEN ER I
LD TR0
AND K1_TR13_TID_S  ; KURS 1 TRINN 13 TID
ANDNOT K1_TR15_TID_S  ; KURS 1 TRINN 15 TID
MOV(021) &12 VST80_K1_TRINN_NR  ; ANGIR VASKETRINN SOM VASKEN ER I
LD TR0
AND K1_TR15_TID_S  ; KURS 1 TRINN 15 TID
ANDNOT K1_TR16_TID_S  ; KURS 1 TRINN 16 TID
MOV(021) &13 VST80_K1_TRINN_NR  ; ANGIR VASKETRINN SOM VASKEN ER I
LD TR0
AND K1_TR16_TID_S  ; KURS 1 TRINN 16 TID
ANDNOT K1_TR17_TID_S  ; KURS 1 TRINN 17 TID
MOV(021) &14 VST80_K1_TRINN_NR  ; ANGIR VASKETRINN SOM VASKEN ER I
LD TR0
AND K1_TR17_TID_S  ; KURS 1 TRINN 17 TID
ANDNOT K1_TR18_TID_S  ; KURS 1 TRINN 18 TID
MOV(021) &15 VST80_K1_TRINN_NR  ; ANGIR VASKETRINN SOM VASKEN ER I

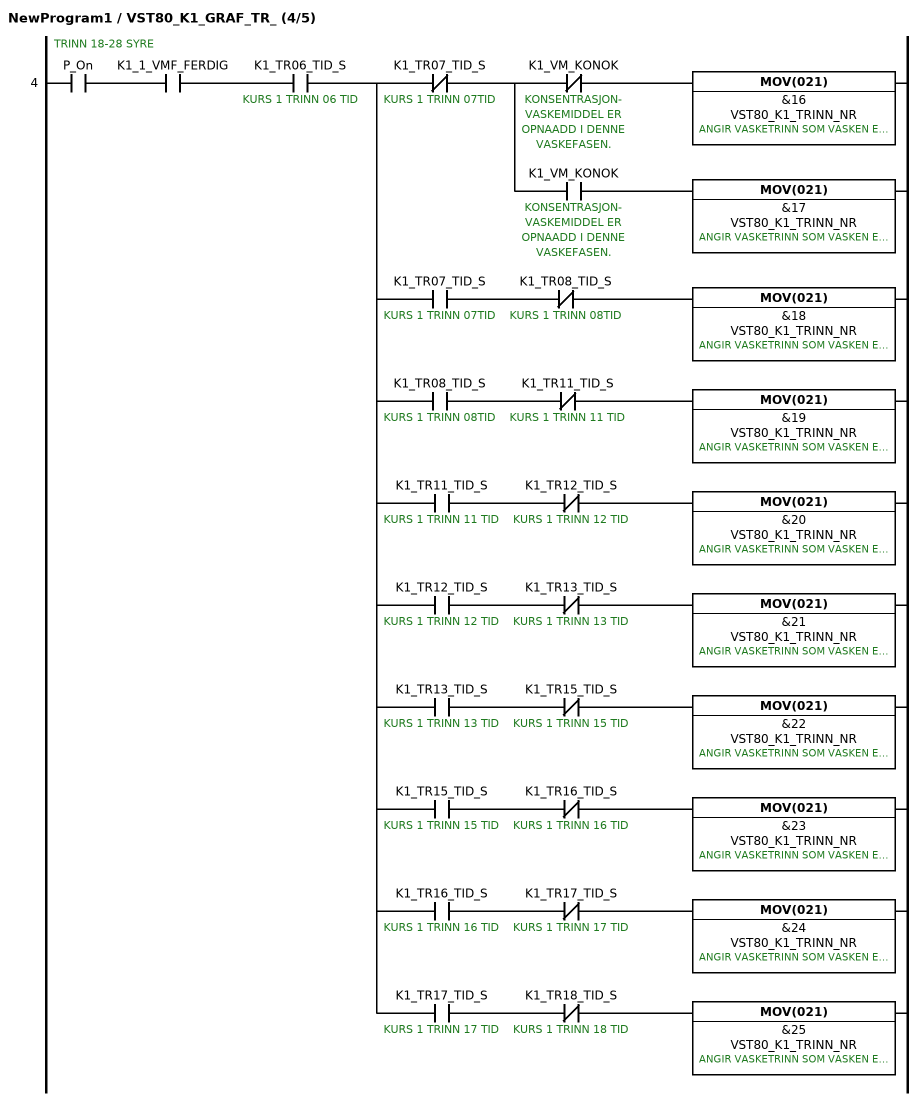
; rung 4: TRINN 18-28 SYRE
LD P_On
AND K1_1_VMF_FERDIG
AND K1_TR06_TID_S  ; KURS 1 TRINN 06 TID
OUT TR0
ANDNOT K1_TR07_TID_S  ; KURS 1 TRINN 07TID
OUT TR1
ANDNOT K1_VM_KONOK  ; KONSENTRASJON-VASKEMIDDEL ER OPNAADD I DENNE VASKEFASEN.
MOV(021) &16 VST80_K1_TRINN_NR  ; ANGIR VASKETRINN SOM VASKEN ER I
LD TR1
AND K1_VM_KONOK  ; KONSENTRASJON-VASKEMIDDEL ER OPNAADD I DENNE VASKEFASEN.
MOV(021) &17 VST80_K1_TRINN_NR  ; ANGIR VASKETRINN SOM VASKEN ER I
LD TR0
AND K1_TR07_TID_S  ; KURS 1 TRINN 07TID
ANDNOT K1_TR08_TID_S  ; KURS 1 TRINN 08TID
MOV(021) &18 VST80_K1_TRINN_NR  ; ANGIR VASKETRINN SOM VASKEN ER I
LD TR0
AND K1_TR08_TID_S  ; KURS 1 TRINN 08TID
ANDNOT K1_TR11_TID_S  ; KURS 1 TRINN 11 TID
MOV(021) &19 VST80_K1_TRINN_NR  ; ANGIR VASKETRINN SOM VASKEN ER I
LD TR0
AND K1_TR11_TID_S  ; KURS 1 TRINN 11 TID
ANDNOT K1_TR12_TID_S  ; KURS 1 TRINN 12 TID
MOV(021) &20 VST80_K1_TRINN_NR  ; ANGIR VASKETRINN SOM VASKEN ER I
LD TR0
AND K1_TR12_TID_S  ; KURS 1 TRINN 12 TID
ANDNOT K1_TR13_TID_S  ; KURS 1 TRINN 13 TID
MOV(021) &21 VST80_K1_TRINN_NR  ; ANGIR VASKETRINN SOM VASKEN ER I
LD TR0
AND K1_TR13_TID_S  ; KURS 1 TRINN 13 TID
ANDNOT K1_TR15_TID_S  ; KURS 1 TRINN 15 TID
MOV(021) &22 VST80_K1_TRINN_NR  ; ANGIR VASKETRINN SOM VASKEN ER I
LD TR0
AND K1_TR15_TID_S  ; KURS 1 TRINN 15 TID
ANDNOT K1_TR16_TID_S  ; KURS 1 TRINN 16 TID
MOV(021) &23 VST80_K1_TRINN_NR  ; ANGIR VASKETRINN SOM VASKEN ER I
LD TR0
AND K1_TR16_TID_S  ; KURS 1 TRINN 16 TID
ANDNOT K1_TR17_TID_S  ; KURS 1 TRINN 17 TID
MOV(021) &24 VST80_K1_TRINN_NR  ; ANGIR VASKETRINN SOM VASKEN ER I
LD TR0
AND K1_TR17_TID_S  ; KURS 1 TRINN 17 TID
ANDNOT K1_TR18_TID_S  ; KURS 1 TRINN 18 TID
MOV(021) &25 VST80_K1_TRINN_NR  ; ANGIR VASKETRINN SOM VASKEN ER I

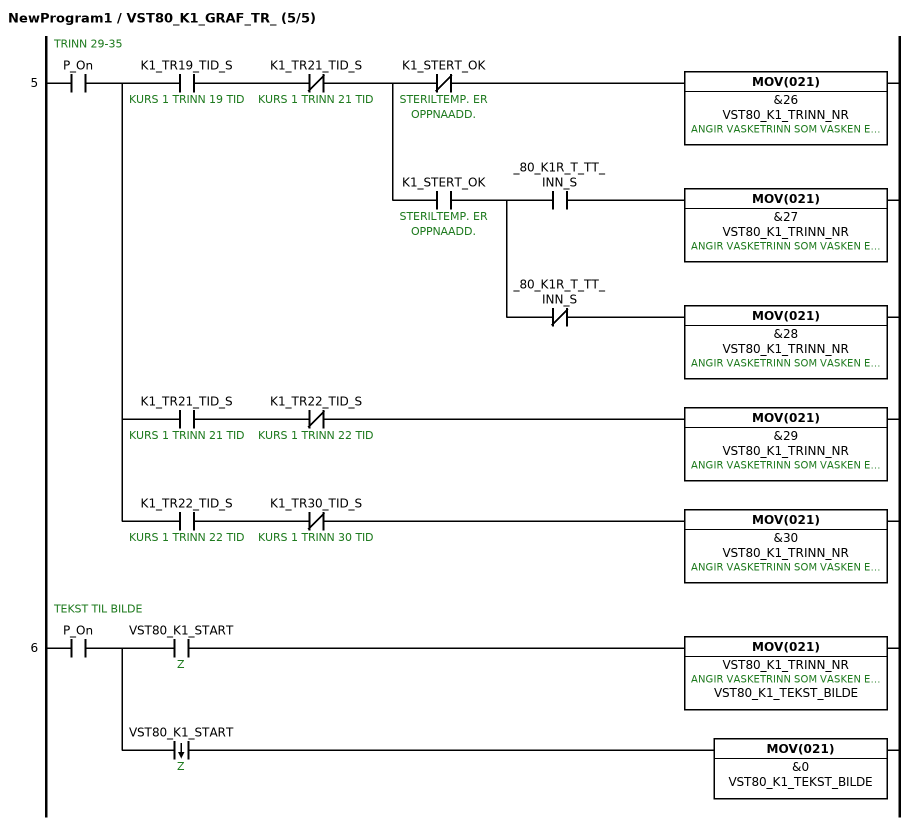
; rung 5: TRINN 29-35
LD P_On
OUT TR0
AND K1_TR19_TID_S  ; KURS 1 TRINN 19 TID
ANDNOT K1_TR21_TID_S  ; KURS 1 TRINN 21 TID
OUT TR1
ANDNOT K1_STERT_OK  ; STERILTEMP. ER OPPNAADD.
MOV(021) &26 VST80_K1_TRINN_NR  ; ANGIR VASKETRINN SOM VASKEN ER I
LD TR1
AND K1_STERT_OK  ; STERILTEMP. ER OPPNAADD.
OUT TR1
AND _80_K1R_T_TT_INN_S
MOV(021) &27 VST80_K1_TRINN_NR  ; ANGIR VASKETRINN SOM VASKEN ER I
LD TR1
ANDNOT _80_K1R_T_TT_INN_S
MOV(021) &28 VST80_K1_TRINN_NR  ; ANGIR VASKETRINN SOM VASKEN ER I
LD TR0
AND K1_TR21_TID_S  ; KURS 1 TRINN 21 TID
ANDNOT K1_TR22_TID_S  ; KURS 1 TRINN 22 TID
MOV(021) &29 VST80_K1_TRINN_NR  ; ANGIR VASKETRINN SOM VASKEN ER I
LD TR0
AND K1_TR22_TID_S  ; KURS 1 TRINN 22 TID
ANDNOT K1_TR30_TID_S  ; KURS 1 TRINN 30 TID
MOV(021) &30 VST80_K1_TRINN_NR  ; ANGIR VASKETRINN SOM VASKEN ER I
; rung 6: TEKST TIL BILDE
LD P_On
OUT TR0
AND VST80_K1_START  ; Z
MOV(021) VST80_K1_TRINN_NR VST80_K1_TEKST_BILDE  ; ANGIR VASKETRINN SOM VASKEN ER I
LD TR0
%AND VST80_K1_START  ; Z
MOV(021) &0 VST80_K1_TEKST_BILDE
; rung 7: Ingen_kommentar_funnet

### Section VST80_K1_ANALOGSIGN_INN

